// ---- DUTs/IO/Topology/Term_294_EK1100_DFE2A59E.TcDUT
{attribute 'GeneratedUsingTerminal: EK1100-0000-0018'}
{attribute addProperty BoxType "EK1100-0000-0018"}
{attribute addProperty Id "Term_300_EL1809EL1809_32157CFD20Term_304_EL2008EL2008_E2806B9511Term_305_EL2008EL2008_E2806B9511"}
{attribute addProperty CRC "3756172702"}
{attribute addProperty Size "42"}
{attribute addProperty Name "Term 294 (EK1100)"}
TYPE Term_294_EK1100_DFE2A59E EXTENDS EK1100_1FC0878B :
STRUCT
    {attribute addProperty Name "Term 300 (EL1809)"}
    {attribute addProperty PreviousPort "Term 294 (EK1100) : B"}
    {attribute addProperty SyncUnit "default"}
    Term_300_EL1809 : EL1809_32157CFD;
    {attribute addProperty Name "Term 304 (EL2008)"}
    {attribute addProperty PreviousPort "Term 300 (EL1809) : B"}
    {attribute addProperty SyncUnit "default"}
    Term_304_EL2008 : EL2008_E2806B95;
    {attribute addProperty Name "Term 305 (EL2008)"}
    {attribute addProperty PreviousPort "Term 304 (EL2008) : B"}
    {attribute addProperty SyncUnit "default"}
    Term_305_EL2008 : EL2008_E2806B95;
END_STRUCT
END_TYPE

// ---- DUTs/IO/Topology/Term_331_EK1100_B9C4E092.TcDUT
{attribute 'GeneratedUsingTerminal: EK1100-0000-0018'}
{attribute addProperty BoxType "EK1100-0000-0018"}
{attribute addProperty Id "Term_332_EL1809EL1809_32157CFD20"}
{attribute addProperty CRC "3116687506"}
{attribute addProperty Size "20"}
{attribute addProperty Name "Term 331 (EK1100)"}
TYPE Term_331_EK1100_B9C4E092 EXTENDS EK1100_1FC0878B :
STRUCT
    {attribute addProperty Name "Term 332 (EL1809)"}
    {attribute addProperty PreviousPort "Term 331 (EK1100) : B"}
    {attribute addProperty SyncUnit "default"}
    Term_332_EL1809 : EL1809_32157CFD;
END_STRUCT
END_TYPE

// ---- DUTs/IO/Topology/Term_333_EK1100_1D6F2042.TcDUT
{attribute 'GeneratedUsingTerminal: EK1100-0000-0018'}
{attribute addProperty BoxType "EK1100-0000-0018"}
{attribute addProperty Id "Term_334_EL1809EL1809_32157CFD20"}
{attribute addProperty CRC "493822018"}
{attribute addProperty Size "20"}
{attribute addProperty Name "Term 333 (EK1100)"}
TYPE Term_333_EK1100_1D6F2042 EXTENDS EK1100_1FC0878B :
STRUCT
    {attribute addProperty Name "Term 334 (EL1809)"}
    {attribute addProperty PreviousPort "Term 333 (EK1100) : B"}
    {attribute addProperty SyncUnit "default"}
    Term_334_EL1809 : EL1809_32157CFD;
END_STRUCT
END_TYPE

// ---- DUTs/IO/Topology/Term_330_EK1122_0EDE60FE.TcDUT
{attribute 'GeneratedUsingTerminal: EK1122-0000-0018'}
{attribute addProperty BoxType "EK1122-0000-0018"}
{attribute addProperty Id "Term_331_EK1100Term_331_EK1100_B9C4E09220Term_333_EK1100Term_333_EK1100_1D6F204220"}
{attribute addProperty CRC "249454846"}
{attribute addProperty Size "40"}
{attribute addProperty Name "Term 330 (EK1122)"}
TYPE Term_330_EK1122_0EDE60FE EXTENDS EK1122_1FC0878B :
STRUCT
    {attribute addProperty Name "Term 331 (EK1100)"}
    {attribute addProperty PreviousPort "Term 330 (EK1122) : D"}
    {attribute addProperty SyncUnit "default"}
    Term_331_EK1100 : Term_331_EK1100_B9C4E092;
    {attribute addProperty Name "Term 333 (EK1100)"}
    {attribute addProperty PreviousPort "Term 331 (EK1100) : C"}
    {attribute addProperty SyncUnit "default"}
    Term_333_EK1100 : Term_333_EK1100_1D6F2042;
END_STRUCT
END_TYPE

// ---- DUTs/IO/Topology/Term_307_EK1100_EB8FAA41.TcDUT
{attribute 'GeneratedUsingTerminal: EK1100-0000-0018'}
{attribute addProperty BoxType "EK1100-0000-0018"}
{attribute addProperty Id "Term_330_EK1122Term_330_EK1122_0EDE60FE40Term_335_EL2008EL2008_E2806B9511Term_336_EL2008EL2008_E2806B9511"}
{attribute addProperty CRC "3952060993"}
{attribute addProperty Size "62"}
{attribute addProperty Name "Term 307 (EK1100)"}
TYPE Term_307_EK1100_EB8FAA41 EXTENDS EK1100_1FC0878B :
STRUCT
    {attribute addProperty Name "Term 330 (EK1122)"}
    {attribute addProperty PreviousPort "Term 307 (EK1100) : B"}
    {attribute addProperty SyncUnit "default"}
    Term_330_EK1122 : Term_330_EK1122_0EDE60FE;
    {attribute addProperty Name "Term 335 (EL2008)"}
    {attribute addProperty PreviousPort "Term 330 (EK1122) : C"}
    {attribute addProperty SyncUnit "default"}
    Term_335_EL2008 : EL2008_E2806B95;
    {attribute addProperty Name "Term 336 (EL2008)"}
    {attribute addProperty PreviousPort "Term 335 (EL2008) : B"}
    {attribute addProperty SyncUnit "default"}
    Term_336_EL2008 : EL2008_E2806B95;
END_STRUCT
END_TYPE

// ---- DUTs/IO/Topology/Term_288_EK1122_18F8921F.TcDUT
{attribute 'GeneratedUsingTerminal: EK1122-0000-0018'}
{attribute addProperty BoxType "EK1122-0000-0018"}
{attribute addProperty Id "Term_289_EK1100Term_289_EK1100_9C677E5049Term_294_EK1100Term_294_EK1100_DFE2A59E42Term_307_EK1100Term_307_EK1100_EB8FAA4162"}
{attribute addProperty CRC "418943519"}
{attribute addProperty Size "153"}
{attribute addProperty Name "Term 288 (EK1122)"}
TYPE Term_288_EK1122_18F8921F EXTENDS EK1122_1FC0878B :
STRUCT
    {attribute addProperty Name "Term 289 (EK1100)"}
    {attribute addProperty PreviousPort "Term 288 (EK1122) : D"}
    {attribute addProperty SyncUnit "default"}
    Term_289_EK1100 : Term_289_EK1100_9C677E50;
    {attribute addProperty Name "Term 294 (EK1100)"}
    {attribute addProperty PreviousPort "Term 289 (EK1100) : C"}
    {attribute addProperty SyncUnit "default"}
    Term_294_EK1100 : Term_294_EK1100_DFE2A59E;
    {attribute addProperty Name "Term 307 (EK1100)"}
    {attribute addProperty PreviousPort "Term 294 (EK1100) : C"}
    {attribute addProperty SyncUnit "default"}
    Term_307_EK1100 : Term_307_EK1100_EB8FAA41;
END_STRUCT
END_TYPE

// ---- DUTs/IO/Topology/Term_146_EK1100_439F5464.TcDUT
{attribute 'GeneratedUsingTerminal: EK1100-0000-0018'}
{attribute addProperty BoxType "EK1100-0000-0018"}
{attribute addProperty Id "Term_147_EK1122Term_147_EK1122_CA6A5D16124Term_186_EK1122Term_186_EK1122_75C79D52124Term_148_EL1809EL1809_32157CFD20Term_149_EL1809EL1809_32157CFD20Term_150_EL1809EL1809_32157CFD20Term_151_EL1809EL1809_32157CFD20Term_152_EL1809EL1809_32157CFD20Term_288_EK1122Term_288_EK1122_18F8921F153Term_1158_EL2008EL2008_E2806B9511Term_1159_EL2008EL2008_E2806B9511Term_1160_EL2008EL2008_E2806B9511Term_1161_EL2008EL2008_E2806B9511Term_1162_EL2008EL2008_E2806B9511Term_1163_EL2008EL2008_E2806B9511"}
{attribute addProperty CRC "1134515300"}
{attribute addProperty Size "567"}
{attribute addProperty Name "Term 146 (EK1100)"}
TYPE Term_146_EK1100_439F5464 EXTENDS EK1100_1FC0878B :
STRUCT
    {attribute addProperty Name "Term 147 (EK1122)"}
    {attribute addProperty PreviousPort "Term 146 (EK1100) : B"}
    {attribute addProperty SyncUnit "default"}
    Term_147_EK1122 : Term_147_EK1122_CA6A5D16;
    {attribute addProperty Name "Term 186 (EK1122)"}
    {attribute addProperty PreviousPort "Term 147 (EK1122) : C"}
    {attribute addProperty SyncUnit "default"}
    Term_186_EK1122 : Term_186_EK1122_75C79D52;
    {attribute addProperty Name "Term 148 (EL1809)"}
    {attribute addProperty PreviousPort "Term 186 (EK1122) : C"}
    {attribute addProperty SyncUnit "default"}
    Term_148_EL1809 : EL1809_32157CFD;
    {attribute addProperty Name "Term 149 (EL1809)"}
    {attribute addProperty PreviousPort "Term 148 (EL1809) : B"}
    {attribute addProperty SyncUnit "default"}
    Term_149_EL1809 : EL1809_32157CFD;
    {attribute addProperty Name "Term 150 (EL1809)"}
    {attribute addProperty PreviousPort "Term 149 (EL1809) : B"}
    {attribute addProperty SyncUnit "default"}
    Term_150_EL1809 : EL1809_32157CFD;
    {attribute addProperty Name "Term 151 (EL1809)"}
    {attribute addProperty PreviousPort "Term 150 (EL1809) : B"}
    {attribute addProperty SyncUnit "default"}
    Term_151_EL1809 : EL1809_32157CFD;
    {attribute addProperty Name "Term 152 (EL1809)"}
    {attribute addProperty PreviousPort "Term 151 (EL1809) : B"}
    {attribute addProperty SyncUnit "default"}
    Term_152_EL1809 : EL1809_32157CFD;
    {attribute addProperty Name "Term 288 (EK1122)"}
    {attribute addProperty PreviousPort "Term 152 (EL1809) : B"}
    {attribute addProperty SyncUnit "default"}
    Term_288_EK1122 : Term_288_EK1122_18F8921F;
    {attribute addProperty Name "Term 1158 (EL2008)"}
    {attribute addProperty PreviousPort "Term 288 (EK1122) : C"}
    {attribute addProperty SyncUnit "default"}
    Term_1158_EL2008 : EL2008_E2806B95;
    {attribute addProperty Name "Term 1159 (EL2008)"}
    {attribute addProperty PreviousPort "Term 1158 (EL2008) : B"}
    {attribute addProperty SyncUnit "default"}
    Term_1159_EL2008 : EL2008_E2806B95;
    {attribute addProperty Name "Term 1160 (EL2008)"}
    {attribute addProperty PreviousPort "Term 1159 (EL2008) : B"}
    {attribute addProperty SyncUnit "default"}
    Term_1160_EL2008 : EL2008_E2806B95;
    {attribute addProperty Name "Term 1161 (EL2008)"}
    {attribute addProperty PreviousPort "Term 1160 (EL2008) : B"}
    {attribute addProperty SyncUnit "default"}
    Term_1161_EL2008 : EL2008_E2806B95;
    {attribute addProperty Name "Term 1162 (EL2008)"}
    {attribute addProperty PreviousPort "Term 1161 (EL2008) : B"}
    {attribute addProperty SyncUnit "default"}
    Term_1162_EL2008 : EL2008_E2806B95;
    {attribute addProperty Name "Term 1163 (EL2008)"}
    {attribute addProperty PreviousPort "Term 1162 (EL2008) : B"}
    {attribute addProperty SyncUnit "default"}
    Term_1163_EL2008 : EL2008_E2806B95;
END_STRUCT
END_TYPE

// ---- DUTs/IO/Topology/Device_3_EtherCAT_368E547E.TcDUT
{attribute 'GeneratedUsingTerminal: IODEVICETYPE_ETHERCATPROT'}
{attribute addProperty BoxType "IODEVICETYPE_ETHERCATPROT"}
{attribute addProperty Id "Term_146_EK1100Term_146_EK1100_439F5464567SyncUnitsSyncUnits_C3A34B5018InputsInputs_A65FACA410OutputsOutputs_23C0ED1D6InfoDataInfoData_84133AC922"}
{attribute addProperty CRC "915297406"}
{attribute addProperty Size "623"}
{attribute addProperty Name "Device 3 (EtherCAT)"}
TYPE Device_3_EtherCAT_368E547E EXTENDS TcoIo.EtcMasterBase_62654B43 :
STRUCT
    {attribute addProperty Name "Term 146 (EK1100)"}
    {attribute addProperty PreviousPort "Device 3 (EtherCAT) : Master"}
    {attribute addProperty SyncUnit "default"}
    Term_146_EK1100 : Term_146_EK1100_439F5464;
    {attribute addProperty Name "SyncUnits"}
    SyncUnits : SyncUnits_C3A34B50;
    {attribute addProperty Name "Inputs"}
    Inputs : TcoIo.Inputs_A65FACA4;
    {attribute addProperty Name "Outputs"}
    Outputs : TcoIo.Outputs_23C0ED1D;
    {attribute addProperty Name "InfoData"}
    InfoData : TcoIo.InfoData_84133AC9;
END_STRUCT
END_TYPE

// ---- DUTs/IO/Topology/R1_A2_EC_EK1122_F4361AFD.TcDUT
{attribute 'GeneratedUsingTerminal: EK1122-0000-0018'}
{attribute addProperty BoxType "EK1122-0000-0018"}
{attribute addProperty Id "Servo_A10_1_AX5106_0000_0203AX5106_1BD22F5129Servo_A10_2_AX5106_0000_0203AX5106_1BD22F5129Servo_A10_3_AX5106_0000_0203AX5106_1BD22F5129"}
{attribute addProperty CRC "4097186557"}
{attribute addProperty Size "87"}
{attribute addProperty Name "R1_A2_EC (EK1122)"}
TYPE R1_A2_EC_EK1122_F4361AFD EXTENDS EK1122_1FC0878B :
STRUCT
    {attribute addProperty Name "Servo_A10_1 (AX5106-0000-0203)"}
    {attribute addProperty PreviousPort "R1_A2_EC (EK1122) : D"}
    {attribute addProperty SyncUnit "default"}
    Servo_A10_1_AX5106_0000_0203 : AX5106_1BD22F51;
    {attribute addProperty Name "Servo_A10_2 (AX5106-0000-0203)"}
    {attribute addProperty PreviousPort "Servo_A10_1 (AX5106-0000-0203) : B"}
    {attribute addProperty SyncUnit "default"}
    Servo_A10_2_AX5106_0000_0203 : AX5106_1BD22F51;
    {attribute addProperty Name "Servo_A10_3 (AX5106-0000-0203)"}
    {attribute addProperty PreviousPort "Servo_A10_2 (AX5106-0000-0203) : B"}
    {attribute addProperty SyncUnit "default"}
    Servo_A10_3_AX5106_0000_0203 : AX5106_1BD22F51;
END_STRUCT
END_TYPE

// ---- DUTs/IO/Topology/R1_A3_EC_EK1122_981C12E1.TcDUT
{attribute 'GeneratedUsingTerminal: EK1122-0000-0018'}
{attribute addProperty BoxType "EK1122-0000-0018"}
{attribute addProperty Id "VI_2_AES_D_BC_ECAT_xAES_A3B0707168VI_4_AES_D_BC_ECAT_xAES_A3B0707168"}
{attribute addProperty CRC "2551976673"}
{attribute addProperty Size "136"}
{attribute addProperty Name "R1_A3_EC (EK1122)"}
TYPE R1_A3_EC_EK1122_981C12E1 EXTENDS EK1122_1FC0878B :
STRUCT
    {attribute addProperty Name "VI-2 (AES-D-BC-ECAT)"}
    {attribute addProperty PreviousPort "R1_A3_EC (EK1122) : D"}
    {attribute addProperty SyncUnit "default"}
    VI_2_AES_D_BC_ECAT_x : AES_A3B07071;
    {attribute addProperty Name "VI-4 (AES-D-BC-ECAT)"}
    {attribute addProperty PreviousPort "R1_A3_EC (EK1122) : B"}
    {attribute addProperty SyncUnit "default"}
    VI_4_AES_D_BC_ECAT_x : AES_A3B07071;
END_STRUCT
END_TYPE

// ---- DUTs/IO/Topology/R1_A4_X1_EK1100_C601B400.TcDUT
{attribute 'GeneratedUsingTerminal: EK1100-0000-0018'}
{attribute addProperty BoxType "EK1100-0000-0018"}
{attribute addProperty Id "R1_A4_X1_PN_EL6631EL6631_A0EC075C2R1_A4_X1_IA1_EL1809EL1809_32157CFD20R1_A4_X1_IA2_EL1809EL1809_32157CFD20R1_A4_X1_IA3_EL1809EL1809_32157CFD20R1_A4_X1_IA4_EL1809EL1809_32157CFD20R1_A4_X1_QA1_EL2809EL2809_2B6483BD19R1_A4_X1_QA2_EL2809EL2809_2B6483BD19R1_A4_X1_QA3_EL2809EL2809_2B6483BD19R1_A4_X1_EndTerminal_EL9010EL9010_D29C20850"}
{attribute addProperty CRC "3322000384"}
{attribute addProperty Size "139"}
{attribute addProperty Name "R1_A4_X1 (EK1100)"}
TYPE R1_A4_X1_EK1100_C601B400 EXTENDS EK1100_1FC0878B :
STRUCT
    {attribute addProperty Name "R1_A4_X1_PN (EL6631)"}
    {attribute addProperty PreviousPort "R1_A4_X1 (EK1100) : B"}
    {attribute addProperty SyncUnit "N10"}
    R1_A4_X1_PN_EL6631 : EL6631_A0EC075C;
    {attribute addProperty Name "R1_A4_X1_IA1 (EL1809)"}
    {attribute addProperty PreviousPort "R1_A4_X1_PN (EL6631) : B"}
    {attribute addProperty SyncUnit "N10"}
    R1_A4_X1_IA1_EL1809 : EL1809_32157CFD;
    {attribute addProperty Name "R1_A4_X1_IA2 (EL1809)"}
    {attribute addProperty PreviousPort "R1_A4_X1_IA1 (EL1809) : B"}
    {attribute addProperty SyncUnit "N10"}
    R1_A4_X1_IA2_EL1809 : EL1809_32157CFD;
    {attribute addProperty Name "R1_A4_X1_IA3 (EL1809)"}
    {attribute addProperty PreviousPort "R1_A4_X1_IA2 (EL1809) : B"}
    {attribute addProperty SyncUnit "N10"}
    R1_A4_X1_IA3_EL1809 : EL1809_32157CFD;
    {attribute addProperty Name "R1_A4_X1_IA4 (EL1809)"}
    {attribute addProperty PreviousPort "R1_A4_X1_IA3 (EL1809) : B"}
    {attribute addProperty SyncUnit "N10"}
    R1_A4_X1_IA4_EL1809 : EL1809_32157CFD;
    {attribute addProperty Name "R1_A4_X1_QA1 (EL2809)"}
    {attribute addProperty PreviousPort "R1_A4_X1_IA4 (EL1809) : B"}
    {attribute addProperty SyncUnit "N10"}
    R1_A4_X1_QA1_EL2809 : EL2809_2B6483BD;
    {attribute addProperty Name "R1_A4_X1_QA2 (EL2809)"}
    {attribute addProperty PreviousPort "R1_A4_X1_QA1 (EL2809) : B"}
    {attribute addProperty SyncUnit "N10"}
    R1_A4_X1_QA2_EL2809 : EL2809_2B6483BD;
    {attribute addProperty Name "R1_A4_X1_QA3 (EL2809)"}
    {attribute addProperty PreviousPort "R1_A4_X1_QA2 (EL2809) : B"}
    {attribute addProperty SyncUnit "N10"}
    R1_A4_X1_QA3_EL2809 : EL2809_2B6483BD;
    {attribute addProperty Name "R1_A4_X1_EndTerminal (EL9010)"}
    {attribute addProperty PreviousPort "R1_A4_X1_QA3 (EL2809) : B"}
    {attribute addProperty SyncUnit "default"}
    R1_A4_X1_EndTerminal_EL9010 : EL9010_D29C2085;
END_STRUCT
END_TYPE

// ---- DUTs/IO/Topology/R1_A4_X2_A2_EK1122_39ABCC27.TcDUT
{attribute 'GeneratedUsingTerminal: EK1122-0000-0018'}
{attribute addProperty BoxType "EK1122-0000-0018"}
{attribute addProperty Id "R1_A4_X2_A2_VI1_AES_D_BC_ECAT_xAES_B47A261080REX_350_IMecat_xIMecat_x_75C6CB6B170"}
{attribute addProperty CRC "967560231"}
{attribute addProperty Size "250"}
{attribute addProperty Name "R1_A4_X2_A2 (EK1122)"}
TYPE R1_A4_X2_A2_EK1122_39ABCC27 EXTENDS EK1122_1FC0878B :
STRUCT
    {attribute addProperty Name "R1_A4_X2_A2_VI1 (AES-D-BC-ECAT)"}
    {attribute addProperty PreviousPort "R1_A4_X2_A2 (EK1122) : D"}
    {attribute addProperty SyncUnit "S10"}
    R1_A4_X2_A2_VI1_AES_D_BC_ECAT_x : AES_B47A2610;
    {attribute addProperty Name "REX_350 (IMecat)"}
    {attribute addProperty PreviousPort "R1_A4_X2_A2 (EK1122) : B"}
    {attribute addProperty SyncUnit "default"}
    REX_350_IMecat_x : IMecat_x_75C6CB6B;
END_STRUCT
END_TYPE

// ---- DUTs/IO/Topology/R1_A4_X2_EK1100_6F5FB3BA.TcDUT
{attribute 'GeneratedUsingTerminal: EK1100-0000-0018'}
{attribute addProperty BoxType "EK1100-0000-0018"}
{attribute addProperty Id "R1_A4_X2_A2_EK1122R1_A4_X2_A2_EK1122_39ABCC27250R1_A4_X2_IA1_EL1809EL1809_32157CFD20R1_A4_X2_IA2_EL1809EL1809_32157CFD20R1_A4_X2_IA3_EL1809EL1809_32157CFD20R1_A4_X2_IA4_EL1809EL1809_32157CFD20R1_A4_X2_IA5_EL1809EL1809_32157CFD20R1_A4_X2_QA1_EL2809EL2809_2B6483BD19R1_A4_X2_QA2_EL2809EL2809_2B6483BD19R1_A4_X2_QA3_EL2809EL2809_2B6483BD19R1_A4_X2_EndTerminal_EL9010EL9010_D29C20850"}
{attribute addProperty CRC "1868542906"}
{attribute addProperty Size "407"}
{attribute addProperty Name "R1_A4_X2 (EK1100)"}
TYPE R1_A4_X2_EK1100_6F5FB3BA EXTENDS EK1100_1FC0878B :
STRUCT
    {attribute addProperty Name "R1_A4_X2_A2 (EK1122)"}
    {attribute addProperty PreviousPort "R1_A4_X2 (EK1100) : B"}
    {attribute addProperty SyncUnit "default"}
    R1_A4_X2_A2_EK1122 : R1_A4_X2_A2_EK1122_39ABCC27;
    {attribute addProperty Name "R1_A4_X2_IA1 (EL1809)"}
    {attribute addProperty PreviousPort "R1_A4_X2_A2 (EK1122) : C"}
    {attribute addProperty SyncUnit "S10"}
    R1_A4_X2_IA1_EL1809 : EL1809_32157CFD;
    {attribute addProperty Name "R1_A4_X2_IA2 (EL1809)"}
    {attribute addProperty PreviousPort "R1_A4_X2_IA1 (EL1809) : B"}
    {attribute addProperty SyncUnit "S10"}
    R1_A4_X2_IA2_EL1809 : EL1809_32157CFD;
    {attribute addProperty Name "R1_A4_X2_IA3 (EL1809)"}
    {attribute addProperty PreviousPort "R1_A4_X2_IA2 (EL1809) : B"}
    {attribute addProperty SyncUnit "S10"}
    R1_A4_X2_IA3_EL1809 : EL1809_32157CFD;
    {attribute addProperty Name "R1_A4_X2_IA4 (EL1809)"}
    {attribute addProperty PreviousPort "R1_A4_X2_IA3 (EL1809) : B"}
    {attribute addProperty SyncUnit "S10"}
    R1_A4_X2_IA4_EL1809 : EL1809_32157CFD;
    {attribute addProperty Name "R1_A4_X2_IA5 (EL1809)"}
    {attribute addProperty PreviousPort "R1_A4_X2_IA4 (EL1809) : B"}
    {attribute addProperty SyncUnit "S10"}
    R1_A4_X2_IA5_EL1809 : EL1809_32157CFD;
    {attribute addProperty Name "R1_A4_X2_QA1 (EL2809)"}
    {attribute addProperty PreviousPort "R1_A4_X2_IA5 (EL1809) : B"}
    {attribute addProperty SyncUnit "S10"}
    R1_A4_X2_QA1_EL2809 : EL2809_2B6483BD;
    {attribute addProperty Name "R1_A4_X2_QA2 (EL2809)"}
    {attribute addProperty PreviousPort "R1_A4_X2_QA1 (EL2809) : B"}
    {attribute addProperty SyncUnit "S10"}
    R1_A4_X2_QA2_EL2809 : EL2809_2B6483BD;
    {attribute addProperty Name "R1_A4_X2_QA3 (EL2809)"}
    {attribute addProperty PreviousPort "R1_A4_X2_QA2 (EL2809) : B"}
    {attribute addProperty SyncUnit "S10"}
    R1_A4_X2_QA3_EL2809 : EL2809_2B6483BD;
    {attribute addProperty Name "R1_A4_X2_EndTerminal (EL9010)"}
    {attribute addProperty PreviousPort "R1_A4_X2_QA3 (EL2809) : B"}
    {attribute addProperty SyncUnit "default"}
    R1_A4_X2_EndTerminal_EL9010 : EL9010_D29C2085;
END_STRUCT
END_TYPE

// ---- DUTs/IO/Topology/R1_A4_EC_EK1122_467C5A0B.TcDUT
{attribute 'GeneratedUsingTerminal: EK1122-0000-0018'}
{attribute addProperty BoxType "EK1122-0000-0018"}
{attribute addProperty Id "R1_A4_X1_EK1100R1_A4_X1_EK1100_C601B400139R1_A4_X2_EK1100R1_A4_X2_EK1100_6F5FB3BA407"}
{attribute addProperty CRC "1182554635"}
{attribute addProperty Size "546"}
{attribute addProperty Name "R1_A4_EC (EK1122)"}
TYPE R1_A4_EC_EK1122_467C5A0B EXTENDS EK1122_1FC0878B :
STRUCT
    {attribute addProperty Name "R1_A4_X1 (EK1100)"}
    {attribute addProperty PreviousPort "R1_A4_EC (EK1122) : D"}
    {attribute addProperty SyncUnit "default"}
    R1_A4_X1_EK1100 : R1_A4_X1_EK1100_C601B400;
    {attribute addProperty Name "R1_A4_X2 (EK1100)"}
    {attribute addProperty PreviousPort "R1_A4_EC (EK1122) : B"}
    {attribute addProperty SyncUnit "default"}
    R1_A4_X2_EK1100 : R1_A4_X2_EK1100_6F5FB3BA;
END_STRUCT
END_TYPE

// ---- DUTs/IO/Topology/R1_EK1100_4AD22B7B.TcDUT
{attribute 'GeneratedUsingTerminal: EK1100-0000-0018'}
{attribute addProperty BoxType "EK1100-0000-0018"}
{attribute addProperty Id "R1_A2_EC_EK1122R1_A2_EC_EK1122_F4361AFD87R1_A3_EC_EK1122R1_A3_EC_EK1122_981C12E1136R1_A4_EC_EK1122R1_A4_EC_EK1122_467C5A0B546R1_A5_DI_EL1809EL1809_32157CFD20R1_A6_DI_EL1809EL1809_32157CFD20R1_A7_DI_EL1809EL1809_32157CFD20R1_A8_DI_EL1809EL1809_32157CFD20R1_A9_DI_EL1809EL1809_32157CFD20R1_A10_DI_EL1809EL1809_32157CFD20R1_A11_DI_EL1809EL1809_32157CFD20R1_A12_DI_EL1809EL1809_32157CFD20R1_A13_DI_EL1809EL1809_32157CFD20R1_A14_DI_EL1809EL1809_32157CFD20R1_A15_DI_EL1809EL1809_32157CFD20R1_A16_DI_EL1809EL1809_32157CFD20R1_A17_DI_EL1809EL1809_32157CFD20R1_A18_DO_EL2809EL2809_2B6483BD19R1_A19_DO_EL2809EL2809_2B6483BD19R1_A20_DO_EL2809EL2809_2B6483BD19R1_A21_DO_EL2809EL2809_2B6483BD19R1_A22_DO_EL2809EL2809_2B6483BD19R1_A23_DO_EL2809EL2809_2B6483BD19R1_EndTerminal_EL9011EL9011_D65D3D320"}
{attribute addProperty CRC "1255287675"}
{attribute addProperty Size "1143"}
{attribute addProperty Name "R1 (EK1100)"}
TYPE R1_EK1100_4AD22B7B EXTENDS EK1100_1FC0878B :
STRUCT
    {attribute addProperty Name "R1_A2_EC (EK1122)"}
    {attribute addProperty PreviousPort "R1 (EK1100) : B"}
    {attribute addProperty SyncUnit "default"}
    R1_A2_EC_EK1122 : R1_A2_EC_EK1122_F4361AFD;
    {attribute addProperty Name "R1_A3_EC (EK1122)"}
    {attribute addProperty PreviousPort "R1_A2_EC (EK1122) : C"}
    {attribute addProperty SyncUnit "default"}
    R1_A3_EC_EK1122 : R1_A3_EC_EK1122_981C12E1;
    {attribute addProperty Name "R1_A4_EC (EK1122)"}
    {attribute addProperty PreviousPort "R1_A3_EC (EK1122) : C"}
    {attribute addProperty SyncUnit "default"}
    R1_A4_EC_EK1122 : R1_A4_EC_EK1122_467C5A0B;
    {attribute addProperty Name "R1_A5_DI (EL1809)"}
    {attribute addProperty PreviousPort "R1_A4_EC (EK1122) : C"}
    {attribute addProperty SyncUnit "default"}
    R1_A5_DI_EL1809 : EL1809_32157CFD;
    {attribute addProperty Name "R1_A6_DI (EL1809)"}
    {attribute addProperty PreviousPort "R1_A5_DI (EL1809) : B"}
    {attribute addProperty SyncUnit "default"}
    R1_A6_DI_EL1809 : EL1809_32157CFD;
    {attribute addProperty Name "R1_A7_DI (EL1809)"}
    {attribute addProperty PreviousPort "R1_A6_DI (EL1809) : B"}
    {attribute addProperty SyncUnit "default"}
    R1_A7_DI_EL1809 : EL1809_32157CFD;
    {attribute addProperty Name "R1_A8_DI (EL1809)"}
    {attribute addProperty PreviousPort "R1_A7_DI (EL1809) : B"}
    {attribute addProperty SyncUnit "default"}
    R1_A8_DI_EL1809 : EL1809_32157CFD;
    {attribute addProperty Name "R1_A9_DI (EL1809)"}
    {attribute addProperty PreviousPort "R1_A8_DI (EL1809) : B"}
    {attribute addProperty SyncUnit "default"}
    R1_A9_DI_EL1809 : EL1809_32157CFD;
    {attribute addProperty Name "R1_A10_DI (EL1809)"}
    {attribute addProperty PreviousPort "R1_A9_DI (EL1809) : B"}
    {attribute addProperty SyncUnit "default"}
    R1_A10_DI_EL1809 : EL1809_32157CFD;
    {attribute addProperty Name "R1_A11_DI (EL1809)"}
    {attribute addProperty PreviousPort "R1_A10_DI (EL1809) : B"}
    {attribute addProperty SyncUnit "default"}
    R1_A11_DI_EL1809 : EL1809_32157CFD;
    {attribute addProperty Name "R1_A12_DI (EL1809)"}
    {attribute addProperty PreviousPort "R1_A11_DI (EL1809) : B"}
    {attribute addProperty SyncUnit "default"}
    R1_A12_DI_EL1809 : EL1809_32157CFD;
    {attribute addProperty Name "R1_A13_DI (EL1809)"}
    {attribute addProperty PreviousPort "R1_A12_DI (EL1809) : B"}
    {attribute addProperty SyncUnit "default"}
    R1_A13_DI_EL1809 : EL1809_32157CFD;
    {attribute addProperty Name "R1_A14_DI (EL1809)"}
    {attribute addProperty PreviousPort "R1_A13_DI (EL1809) : B"}
    {attribute addProperty SyncUnit "default"}
    R1_A14_DI_EL1809 : EL1809_32157CFD;
    {attribute addProperty Name "R1_A15_DI (EL1809)"}
    {attribute addProperty PreviousPort "R1_A14_DI (EL1809) : B"}
    {attribute addProperty SyncUnit "default"}
    R1_A15_DI_EL1809 : EL1809_32157CFD;
    {attribute addProperty Name "R1_A16_DI (EL1809)"}
    {attribute addProperty PreviousPort "R1_A15_DI (EL1809) : B"}
    {attribute addProperty SyncUnit "default"}
    R1_A16_DI_EL1809 : EL1809_32157CFD;
    {attribute addProperty Name "R1_A17_DI (EL1809)"}
    {attribute addProperty PreviousPort "R1_A16_DI (EL1809) : B"}
    {attribute addProperty SyncUnit "default"}
    R1_A17_DI_EL1809 : EL1809_32157CFD;
    {attribute addProperty Name "R1_A18_DO (EL2809)"}
    {attribute addProperty PreviousPort "R1_A17_DI (EL1809) : B"}
    {attribute addProperty SyncUnit "default"}
    R1_A18_DO_EL2809 : EL2809_2B6483BD;
    {attribute addProperty Name "R1_A19_DO (EL2809)"}
    {attribute addProperty PreviousPort "R1_A18_DO (EL2809) : B"}
    {attribute addProperty SyncUnit "default"}
    R1_A19_DO_EL2809 : EL2809_2B6483BD;
    {attribute addProperty Name "R1_A20_DO (EL2809)"}
    {attribute addProperty PreviousPort "R1_A19_DO (EL2809) : B"}
    {attribute addProperty SyncUnit "default"}
    R1_A20_DO_EL2809 : EL2809_2B6483BD;
    {attribute addProperty Name "R1_A21_DO (EL2809)"}
    {attribute addProperty PreviousPort "R1_A20_DO (EL2809) : B"}
    {attribute addProperty SyncUnit "default"}
    R1_A21_DO_EL2809 : EL2809_2B6483BD;
    {attribute addProperty Name "R1_A22_DO (EL2809)"}
    {attribute addProperty PreviousPort "R1_A21_DO (EL2809) : B"}
    {attribute addProperty SyncUnit "default"}
    R1_A22_DO_EL2809 : EL2809_2B6483BD;
    {attribute addProperty Name "R1_A23_DO (EL2809)"}
    {attribute addProperty PreviousPort "R1_A22_DO (EL2809) : B"}
    {attribute addProperty SyncUnit "default"}
    R1_A23_DO_EL2809 : EL2809_2B6483BD;
    {attribute addProperty Name "R1_EndTerminal (EL9011)"}
    {attribute addProperty PreviousPort "R1_A23_DO (EL2809) : B"}
    {attribute addProperty SyncUnit "default"}
    R1_EndTerminal_EL9011 : EL9011_D65D3D32;
END_STRUCT
END_TYPE

// ---- DUTs/IO/Topology/R2_A2_EC_EK1122_6D3594D4.TcDUT
{attribute 'GeneratedUsingTerminal: EK1122-0000-0018'}
{attribute addProperty BoxType "EK1122-0000-0018"}
{attribute addProperty Id "Servo_A20_2_AX5103_0000_0203AX5103_1BD22F5129VI_3_AES_D_BC_ECAT_xAES_A3B0707168"}
{attribute addProperty CRC "1832228052"}
{attribute addProperty Size "97"}
{attribute addProperty Name "R2_A2_EC (EK1122)"}
TYPE R2_A2_EC_EK1122_6D3594D4 EXTENDS EK1122_1FC0878B :
STRUCT
    {attribute addProperty Name "Servo_A20-2 (AX5103-0000-0203)"}
    {attribute addProperty PreviousPort "R2_A2_EC (EK1122) : D"}
    {attribute addProperty SyncUnit "default"}
    Servo_A20_2_AX5103_0000_0203 : AX5103_1BD22F51;
    {attribute addProperty Name "VI-3 (AES-D-BC-ECAT)"}
    {attribute addProperty PreviousPort "R2_A2_EC (EK1122) : B"}
    {attribute addProperty SyncUnit "default"}
    VI_3_AES_D_BC_ECAT_x : AES_A3B07071;
END_STRUCT
END_TYPE

// ---- DUTs/IO/Topology/R2_EK1100_10D8A594.TcDUT
{attribute 'GeneratedUsingTerminal: EK1100-0000-0018'}
{attribute addProperty BoxType "EK1100-0000-0018"}
{attribute addProperty Id "R2_A2_EC_EK1122R2_A2_EC_EK1122_6D3594D497R2_A3_DI_EL1809EL1809_32157CFD20R2_A4_DI_EL1809EL1809_32157CFD20R2_A5_DI_EL1809EL1809_32157CFD20R2_A6_DI_EL1809EL1809_32157CFD20R2_A7_DI_EL1809EL1809_32157CFD20R2_A8_DI_EL1809EL1809_32157CFD20R2_A9_DI_EL1809EL1809_32157CFD20R2_A10_DI_EL1809EL1809_32157CFD20R2_A11_DC_EL7332EL7332_DFB2BED746R2_A12_DI_EL1809EL1809_32157CFD20R2_A13_DI_EL1809EL1809_32157CFD20R2_A14_DI_EL1809EL1809_32157CFD20R2_A15_DO_EL2809EL2809_2B6483BD19R2_A16_DO_EL2809EL2809_2B6483BD19R2_A17_DO_EL2809EL2809_2B6483BD19R2_A18_DO_EL2809EL2809_2B6483BD19R2_A19_DO_EL2809EL2809_2B6483BD19R2_EndTerminal_EL9011EL9011_D65D3D320"}
{attribute addProperty CRC "282633620"}
{attribute addProperty Size "458"}
{attribute addProperty Name "R2 (EK1100)"}
TYPE R2_EK1100_10D8A594 EXTENDS EK1100_1FC0878B :
STRUCT
    {attribute addProperty Name "R2_A2_EC (EK1122)"}
    {attribute addProperty PreviousPort "R2 (EK1100) : B"}
    {attribute addProperty SyncUnit "default"}
    R2_A2_EC_EK1122 : R2_A2_EC_EK1122_6D3594D4;
    {attribute addProperty Name "R2_A3_DI (EL1809)"}
    {attribute addProperty PreviousPort "R2_A2_EC (EK1122) : C"}
    {attribute addProperty SyncUnit "default"}
    R2_A3_DI_EL1809 : EL1809_32157CFD;
    {attribute addProperty Name "R2_A4_DI (EL1809)"}
    {attribute addProperty PreviousPort "R2_A3_DI (EL1809) : B"}
    {attribute addProperty SyncUnit "default"}
    R2_A4_DI_EL1809 : EL1809_32157CFD;
    {attribute addProperty Name "R2_A5_DI (EL1809)"}
    {attribute addProperty PreviousPort "R2_A4_DI (EL1809) : B"}
    {attribute addProperty SyncUnit "default"}
    R2_A5_DI_EL1809 : EL1809_32157CFD;
    {attribute addProperty Name "R2_A6_DI (EL1809)"}
    {attribute addProperty PreviousPort "R2_A5_DI (EL1809) : B"}
    {attribute addProperty SyncUnit "default"}
    R2_A6_DI_EL1809 : EL1809_32157CFD;
    {attribute addProperty Name "R2_A7_DI (EL1809)"}
    {attribute addProperty PreviousPort "R2_A6_DI (EL1809) : B"}
    {attribute addProperty SyncUnit "default"}
    R2_A7_DI_EL1809 : EL1809_32157CFD;
    {attribute addProperty Name "R2_A8_DI (EL1809)"}
    {attribute addProperty PreviousPort "R2_A7_DI (EL1809) : B"}
    {attribute addProperty SyncUnit "default"}
    R2_A8_DI_EL1809 : EL1809_32157CFD;
    {attribute addProperty Name "R2_A9_DI (EL1809)"}
    {attribute addProperty PreviousPort "R2_A8_DI (EL1809) : B"}
    {attribute addProperty SyncUnit "default"}
    R2_A9_DI_EL1809 : EL1809_32157CFD;
    {attribute addProperty Name "R2_A10_DI (EL1809)"}
    {attribute addProperty PreviousPort "R2_A9_DI (EL1809) : B"}
    {attribute addProperty SyncUnit "default"}
    R2_A10_DI_EL1809 : EL1809_32157CFD;
    {attribute addProperty Name "R2_A11_DC (EL7332)"}
    {attribute addProperty PreviousPort "R2_A10_DI (EL1809) : B"}
    {attribute addProperty SyncUnit "default"}
    R2_A11_DC_EL7332 : EL7332_DFB2BED7;
    {attribute addProperty Name "R2_A12_DI (EL1809)"}
    {attribute addProperty PreviousPort "R2_A11_DC (EL7332) : B"}
    {attribute addProperty SyncUnit "default"}
    R2_A12_DI_EL1809 : EL1809_32157CFD;
    {attribute addProperty Name "R2_A13_DI (EL1809)"}
    {attribute addProperty PreviousPort "R2_A12_DI (EL1809) : B"}
    {attribute addProperty SyncUnit "default"}
    R2_A13_DI_EL1809 : EL1809_32157CFD;
    {attribute addProperty Name "R2_A14_DI (EL1809)"}
    {attribute addProperty PreviousPort "R2_A13_DI (EL1809) : B"}
    {attribute addProperty SyncUnit "default"}
    R2_A14_DI_EL1809 : EL1809_32157CFD;
    {attribute addProperty Name "R2_A15_DO (EL2809)"}
    {attribute addProperty PreviousPort "R2_A14_DI (EL1809) : B"}
    {attribute addProperty SyncUnit "default"}
    R2_A15_DO_EL2809 : EL2809_2B6483BD;
    {attribute addProperty Name "R2_A16_DO (EL2809)"}
    {attribute addProperty PreviousPort "R2_A15_DO (EL2809) : B"}
    {attribute addProperty SyncUnit "default"}
    R2_A16_DO_EL2809 : EL2809_2B6483BD;
    {attribute addProperty Name "R2_A17_DO (EL2809)"}
    {attribute addProperty PreviousPort "R2_A16_DO (EL2809) : B"}
    {attribute addProperty SyncUnit "default"}
    R2_A17_DO_EL2809 : EL2809_2B6483BD;
    {attribute addProperty Name "R2_A18_DO (EL2809)"}
    {attribute addProperty PreviousPort "R2_A17_DO (EL2809) : B"}
    {attribute addProperty SyncUnit "default"}
    R2_A18_DO_EL2809 : EL2809_2B6483BD;
    {attribute addProperty Name "R2_A19_DO (EL2809)"}
    {attribute addProperty PreviousPort "R2_A18_DO (EL2809) : B"}
    {attribute addProperty SyncUnit "default"}
    R2_A19_DO_EL2809 : EL2809_2B6483BD;
    {attribute addProperty Name "R2_EndTerminal (EL9011)"}
    {attribute addProperty PreviousPort "R2_A19_DO (EL2809) : B"}
    {attribute addProperty SyncUnit "default"}
    R2_EndTerminal_EL9011 : EL9011_D65D3D32;
END_STRUCT
END_TYPE

// ---- DUTs/IO/Topology/R3_A2_EC_EK1122_9D59CDC8.TcDUT
{attribute 'GeneratedUsingTerminal: EK1122-0000-0018'}
{attribute addProperty BoxType "EK1122-0000-0018"}
{attribute addProperty Id "R3_FESTO_CMMP_AS_V4p0_CiA402CMMP_93B92D5237VI_1_AES_D_BC_ECAT_xAES_A3B0707168"}
{attribute addProperty CRC "2639908296"}
{attribute addProperty Size "105"}
{attribute addProperty Name "R3_A2_EC (EK1122)"}
TYPE R3_A2_EC_EK1122_9D59CDC8 EXTENDS EK1122_1FC0878B :
STRUCT
    {attribute addProperty Name "R3_FESTO (CMMP-AS V4p0 CiA402)"}
    {attribute addProperty PreviousPort "R3_A2_EC (EK1122) : D"}
    {attribute addProperty SyncUnit "default"}
    R3_FESTO_CMMP_AS_V4p0_CiA402 : CMMP_93B92D52;
    {attribute addProperty Name "VI-1 (AES-D-BC-ECAT)"}
    {attribute addProperty PreviousPort "R3_A2_EC (EK1122) : B"}
    {attribute addProperty SyncUnit "default"}
    VI_1_AES_D_BC_ECAT_x : AES_A3B07071;
END_STRUCT
END_TYPE

// ---- DUTs/IO/Topology/R3_EK1100_C7887D6C.TcDUT
{attribute 'GeneratedUsingTerminal: EK1100-0000-0018'}
{attribute addProperty BoxType "EK1100-0000-0018"}
{attribute addProperty Id "R3_A2_EC_EK1122R3_A2_EC_EK1122_9D59CDC8105R3_A3_DI_EL1809EL1809_32157CFD20R3_A4_DI_EL1809EL1809_32157CFD20R3_A5_DI_EL1809EL1809_32157CFD20R3_A6_DI_EL1809EL1809_32157CFD20R3_A7_DI_EL1809EL1809_32157CFD20R3_A8_DI_EL1809EL1809_32157CFD20R3_A9_DO_EL2809EL2809_2B6483BD19R3_A10_DO_EL2809EL2809_2B6483BD19R3_EndTerminal_EL9011EL9011_D65D3D320"}
{attribute addProperty CRC "3347610988"}
{attribute addProperty Size "263"}
{attribute addProperty Name "R3 (EK1100)"}
TYPE R3_EK1100_C7887D6C EXTENDS EK1100_1FC0878B :
STRUCT
    {attribute addProperty Name "R3_A2_EC (EK1122)"}
    {attribute addProperty PreviousPort "R3 (EK1100) : B"}
    {attribute addProperty SyncUnit "default"}
    R3_A2_EC_EK1122 : R3_A2_EC_EK1122_9D59CDC8;
    {attribute addProperty Name "R3_A3_DI (EL1809)"}
    {attribute addProperty PreviousPort "R3_A2_EC (EK1122) : C"}
    {attribute addProperty SyncUnit "default"}
    R3_A3_DI_EL1809 : EL1809_32157CFD;
    {attribute addProperty Name "R3_A4_DI (EL1809)"}
    {attribute addProperty PreviousPort "R3_A3_DI (EL1809) : B"}
    {attribute addProperty SyncUnit "default"}
    R3_A4_DI_EL1809 : EL1809_32157CFD;
    {attribute addProperty Name "R3_A5_DI (EL1809)"}
    {attribute addProperty PreviousPort "R3_A4_DI (EL1809) : B"}
    {attribute addProperty SyncUnit "default"}
    R3_A5_DI_EL1809 : EL1809_32157CFD;
    {attribute addProperty Name "R3_A6_DI (EL1809)"}
    {attribute addProperty PreviousPort "R3_A5_DI (EL1809) : B"}
    {attribute addProperty SyncUnit "default"}
    R3_A6_DI_EL1809 : EL1809_32157CFD;
    {attribute addProperty Name "R3_A7_DI (EL1809)"}
    {attribute addProperty PreviousPort "R3_A6_DI (EL1809) : B"}
    {attribute addProperty SyncUnit "default"}
    R3_A7_DI_EL1809 : EL1809_32157CFD;
    {attribute addProperty Name "R3_A8_DI (EL1809)"}
    {attribute addProperty PreviousPort "R3_A7_DI (EL1809) : B"}
    {attribute addProperty SyncUnit "default"}
    R3_A8_DI_EL1809 : EL1809_32157CFD;
    {attribute addProperty Name "R3_A9_DO (EL2809)"}
    {attribute addProperty PreviousPort "R3_A8_DI (EL1809) : B"}
    {attribute addProperty SyncUnit "default"}
    R3_A9_DO_EL2809 : EL2809_2B6483BD;
    {attribute addProperty Name "R3_A10_DO (EL2809)"}
    {attribute addProperty PreviousPort "R3_A9_DO (EL2809) : B"}
    {attribute addProperty SyncUnit "default"}
    R3_A10_DO_EL2809 : EL2809_2B6483BD;
    {attribute addProperty Name "R3_EndTerminal (EL9011)"}
    {attribute addProperty PreviousPort "R3_A10_DO (EL2809) : B"}
    {attribute addProperty SyncUnit "default"}
    R3_EndTerminal_EL9011 : EL9011_D65D3D32;
END_STRUCT
END_TYPE

// ---- DUTs/IO/Topology/RH_A2_X2_EK1100_67419BB1.TcDUT
{attribute 'GeneratedUsingTerminal: EK1100-0000-0018'}
{attribute addProperty BoxType "EK1100-0000-0018"}
{attribute addProperty Id "RH_A2_X2_A2_EL7211_0010EL7211_008D5C9A30RH_A2_X2_A3_EL1809EL1809_32157CFD20RH_A2_X2_A4_EL2809EL2809_2B6483BD19Term_1057_EL9011EL9011_D65D3D320"}
{attribute addProperty CRC "1732352945"}
{attribute addProperty Size "69"}
{attribute addProperty Name "RH_A2_X2 (EK1100)"}
TYPE RH_A2_X2_EK1100_67419BB1 EXTENDS EK1100_1FC0878B :
STRUCT
    {attribute addProperty Name "RH_A2_X2_A2 (EL7211-0010)"}
    {attribute addProperty PreviousPort "RH_A2_X2 (EK1100) : B"}
    {attribute addProperty SyncUnit "RH"}
    RH_A2_X2_A2_EL7211_0010 : EL7211_008D5C9A;
    {attribute addProperty Name "RH_A2_X2_A3 (EL1809)"}
    {attribute addProperty PreviousPort "RH_A2_X2_A2 (EL7211-0010) : B"}
    {attribute addProperty SyncUnit "RH"}
    RH_A2_X2_A3_EL1809 : EL1809_32157CFD;
    {attribute addProperty Name "RH_A2_X2_A4 (EL2809)"}
    {attribute addProperty PreviousPort "RH_A2_X2_A3 (EL1809) : B"}
    {attribute addProperty SyncUnit "RH"}
    RH_A2_X2_A4_EL2809 : EL2809_2B6483BD;
    {attribute addProperty Name "Term 1057 (EL9011)"}
    {attribute addProperty PreviousPort "RH_A2_X2_A4 (EL2809) : B"}
    {attribute addProperty SyncUnit "default"}
    Term_1057_EL9011 : EL9011_D65D3D32;
END_STRUCT
END_TYPE

// ---- DUTs/IO/Topology/RH_A2_EK1122_10728E09.TcDUT
{attribute 'GeneratedUsingTerminal: EK1122-0000-0018'}
{attribute addProperty BoxType "EK1122-0000-0018"}
{attribute addProperty Id "RH_SAFETY_Flexi_Gateway_GETC1Flexi_Gateway_GETC1_429ECB705RH_A2_X2_EK1100RH_A2_X2_EK1100_67419BB169"}
{attribute addProperty CRC "275942921"}
{attribute addProperty Size "74"}
{attribute addProperty Name "RH_A2 (EK1122)"}
TYPE RH_A2_EK1122_10728E09 EXTENDS EK1122_1FC0878B :
STRUCT
    {attribute addProperty Name "RH_SAFETY (Flexi Gateway GETC1)"}
    {attribute addProperty PreviousPort "RH_A2 (EK1122) : D"}
    {attribute addProperty SyncUnit "RH"}
    RH_SAFETY_Flexi_Gateway_GETC1 : Flexi_Gateway_GETC1_429ECB70;
    {attribute addProperty Name "RH_A2_X2 (EK1100)"}
    {attribute addProperty PreviousPort "RH_A2 (EK1122) : B"}
    {attribute addProperty SyncUnit "default"}
    RH_A2_X2_EK1100 : RH_A2_X2_EK1100_67419BB1;
END_STRUCT
END_TYPE

// ---- DUTs/IO/Topology/RH_EK1100_A5940DFE.TcDUT
{attribute 'GeneratedUsingTerminal: EK1100-0000-0018'}
{attribute addProperty BoxType "EK1100-0000-0018"}
{attribute addProperty Id "RH_A2_EK1122RH_A2_EK1122_10728E0974RH_A3_EL6631EL6631_A0EC075C2RH_A4_EL1809EL1809_32157CFD20RH_A5_EL1809EL1809_32157CFD20RH_A6_EL1809EL1809_32157CFD20RH_A7_EL2809EL2809_2B6483BD19RH_A8_EL1809EL1809_32157CFD20RH_A9_EL2809EL2809_2B6483BD19RH_A10_EL2809EL2809_2B6483BD19RH_A11_EL2809EL2809_2B6483BD19RH_EndTerminal_EL9011EL9011_D65D3D320"}
{attribute addProperty CRC "2777943550"}
{attribute addProperty Size "232"}
{attribute addProperty Name "RH (EK1100)"}
TYPE RH_EK1100_A5940DFE EXTENDS EK1100_1FC0878B :
STRUCT
    {attribute addProperty Name "RH_A2 (EK1122)"}
    {attribute addProperty PreviousPort "RH (EK1100) : B"}
    {attribute addProperty SyncUnit "default"}
    RH_A2_EK1122 : RH_A2_EK1122_10728E09;
    {attribute addProperty Name "RH_A3 (EL6631)"}
    {attribute addProperty PreviousPort "RH_A2 (EK1122) : C"}
    {attribute addProperty SyncUnit "RH"}
    RH_A3_EL6631 : EL6631_A0EC075C;
    {attribute addProperty Name "RH_A4 (EL1809)"}
    {attribute addProperty PreviousPort "RH_A3 (EL6631) : B"}
    {attribute addProperty SyncUnit "RH"}
    RH_A4_EL1809 : EL1809_32157CFD;
    {attribute addProperty Name "RH_A5 (EL1809)"}
    {attribute addProperty PreviousPort "RH_A4 (EL1809) : B"}
    {attribute addProperty SyncUnit "RH"}
    RH_A5_EL1809 : EL1809_32157CFD;
    {attribute addProperty Name "RH_A6 (EL1809)"}
    {attribute addProperty PreviousPort "RH_A5 (EL1809) : B"}
    {attribute addProperty SyncUnit "RH"}
    RH_A6_EL1809 : EL1809_32157CFD;
    {attribute addProperty Name "RH_A7 (EL2809)"}
    {attribute addProperty PreviousPort "RH_A6 (EL1809) : B"}
    {attribute addProperty SyncUnit "RH"}
    RH_A7_EL2809 : EL2809_2B6483BD;
    {attribute addProperty Name "RH_A8 (EL1809)"}
    {attribute addProperty PreviousPort "RH_A7 (EL2809) : B"}
    {attribute addProperty SyncUnit "RH"}
    RH_A8_EL1809 : EL1809_32157CFD;
    {attribute addProperty Name "RH_A9 (EL2809)"}
    {attribute addProperty PreviousPort "RH_A8 (EL1809) : B"}
    {attribute addProperty SyncUnit "RH"}
    RH_A9_EL2809 : EL2809_2B6483BD;
    {attribute addProperty Name "RH_A10 (EL2809)"}
    {attribute addProperty PreviousPort "RH_A9 (EL2809) : B"}
    {attribute addProperty SyncUnit "RH"}
    RH_A10_EL2809 : EL2809_2B6483BD;
    {attribute addProperty Name "RH_A11 (EL2809)"}
    {attribute addProperty PreviousPort "RH_A10 (EL2809) : B"}
    {attribute addProperty SyncUnit "RH"}
    RH_A11_EL2809 : EL2809_2B6483BD;
    {attribute addProperty Name "RH_EndTerminal (EL9011)"}
    {attribute addProperty PreviousPort "RH_A11 (EL2809) : B"}
    {attribute addProperty SyncUnit "default"}
    RH_EndTerminal_EL9011 : EL9011_D65D3D32;
END_STRUCT
END_TYPE

// ---- DUTs/IO/Topology/R4_A2_EC_EK1122_254454A1.TcDUT
{attribute 'GeneratedUsingTerminal: EK1122-0000-0018'}
{attribute addProperty BoxType "EK1122-0000-0018"}
{attribute addProperty Id "R4_FESTO_CMMP_AS_V4p0_CiA402CMMP_93B92D5237RH_EK1100RH_EK1100_A5940DFE232"}
{attribute addProperty CRC "625235105"}
{attribute addProperty Size "269"}
{attribute addProperty Name "R4_A2_EC (EK1122)"}
TYPE R4_A2_EC_EK1122_254454A1 EXTENDS EK1122_1FC0878B :
STRUCT
    {attribute addProperty Name "R4_FESTO (CMMP-AS V4p0 CiA402)"}
    {attribute addProperty PreviousPort "R4_A2_EC (EK1122) : D"}
    {attribute addProperty SyncUnit "default"}
    R4_FESTO_CMMP_AS_V4p0_CiA402 : CMMP_93B92D52;
    {attribute addProperty Name "RH (EK1100)"}
    {attribute addProperty PreviousPort "R4_A2_EC (EK1122) : B"}
    {attribute addProperty SyncUnit "default"}
    RH_EK1100 : RH_EK1100_A5940DFE;
END_STRUCT
END_TYPE

// ---- DUTs/IO/Topology/R4_EK1100_46A1248C.TcDUT
{attribute 'GeneratedUsingTerminal: EK1100-0000-0018'}
{attribute addProperty BoxType "EK1100-0000-0018"}
{attribute addProperty Id "R4_A2_EC_EK1122R4_A2_EC_EK1122_254454A1269R4_A3_DI_EL1809EL1809_32157CFD20R4_A4_DI_EL1809EL1809_32157CFD20R4_A5_DI_EL1809EL1809_32157CFD20R4_A6_DI_EL1809EL1809_32157CFD20R4_A7_DI_EL1809EL1809_32157CFD20R4_EndTerminal_EL9011EL9011_D65D3D320"}
{attribute addProperty CRC "1184965772"}
{attribute addProperty Size "369"}
{attribute addProperty Name "R4 (EK1100)"}
TYPE R4_EK1100_46A1248C EXTENDS EK1100_1FC0878B :
STRUCT
    {attribute addProperty Name "R4_A2_EC (EK1122)"}
    {attribute addProperty PreviousPort "R4 (EK1100) : B"}
    {attribute addProperty SyncUnit "default"}
    R4_A2_EC_EK1122 : R4_A2_EC_EK1122_254454A1;
    {attribute addProperty Name "R4_A3_DI (EL1809)"}
    {attribute addProperty PreviousPort "R4_A2_EC (EK1122) : C"}
    {attribute addProperty SyncUnit "default"}
    R4_A3_DI_EL1809 : EL1809_32157CFD;
    {attribute addProperty Name "R4_A4_DI (EL1809)"}
    {attribute addProperty PreviousPort "R4_A3_DI (EL1809) : B"}
    {attribute addProperty SyncUnit "default"}
    R4_A4_DI_EL1809 : EL1809_32157CFD;
    {attribute addProperty Name "R4_A5_DI (EL1809)"}
    {attribute addProperty PreviousPort "R4_A4_DI (EL1809) : B"}
    {attribute addProperty SyncUnit "default"}
    R4_A5_DI_EL1809 : EL1809_32157CFD;
    {attribute addProperty Name "R4_A6_DI (EL1809)"}
    {attribute addProperty PreviousPort "R4_A5_DI (EL1809) : B"}
    {attribute addProperty SyncUnit "default"}
    R4_A6_DI_EL1809 : EL1809_32157CFD;
    {attribute addProperty Name "R4_A7_DI (EL1809)"}
    {attribute addProperty PreviousPort "R4_A6_DI (EL1809) : B"}
    {attribute addProperty SyncUnit "default"}
    R4_A7_DI_EL1809 : EL1809_32157CFD;
    {attribute addProperty Name "R4_EndTerminal (EL9011)"}
    {attribute addProperty PreviousPort "R4_A7_DI (EL1809) : B"}
    {attribute addProperty SyncUnit "default"}
    R4_EndTerminal_EL9011 : EL9011_D65D3D32;
END_STRUCT
END_TYPE

// ---- DUTs/IO/Topology/A2_EK1122_967E4A9C.TcDUT
{attribute 'GeneratedUsingTerminal: EK1122-0000-0018'}
{attribute addProperty BoxType "EK1122-0000-0018"}
{attribute addProperty Id "VI_7_AES_D_BC_ECAT_xAES_A3B0707168"}
{attribute addProperty CRC "2524859036"}
{attribute addProperty Size "68"}
{attribute addProperty Name "A2 (EK1122)"}
TYPE A2_EK1122_967E4A9C EXTENDS EK1122_1FC0878B :
STRUCT
    {attribute addProperty Name "VI-7 (AES-D-BC-ECAT)"}
    {attribute addProperty PreviousPort "A2 (EK1122) : D"}
    {attribute addProperty SyncUnit "default"}
    VI_7_AES_D_BC_ECAT_x : AES_A3B07071;
END_STRUCT
END_TYPE

// ---- DUTs/IO/Topology/R4A_EK1100_48316913.TcDUT
{attribute 'GeneratedUsingTerminal: EK1100-0000-0018'}
{attribute addProperty BoxType "EK1100-0000-0018"}
{attribute addProperty Id "A2_EK1122A2_EK1122_967E4A9C68A3_EL1809EL1809_32157CFD20A4_EL1809EL1809_32157CFD20A5_EL1809EL1809_32157CFD20A6_EL1809EL1809_32157CFD20A7_EL3692EL3692_73B9410052A8_EL3692EL3692_73B9410052A9_EL2008EL2008_E2806B9511A10_EL2008EL2008_E2806B9511R4A_EndTerminal_EL9011EL9011_D65D3D320"}
{attribute addProperty CRC "1211197715"}
{attribute addProperty Size "274"}
{attribute addProperty Name "R4A (EK1100)"}
TYPE R4A_EK1100_48316913 EXTENDS EK1100_1FC0878B :
STRUCT
    {attribute addProperty Name "A2 (EK1122)"}
    {attribute addProperty PreviousPort "R4A (EK1100) : B"}
    {attribute addProperty SyncUnit "default"}
    A2_EK1122 : A2_EK1122_967E4A9C;
    {attribute addProperty Name "A3 (EL1809)"}
    {attribute addProperty PreviousPort "A2 (EK1122) : C"}
    {attribute addProperty SyncUnit "default"}
    A3_EL1809 : EL1809_32157CFD;
    {attribute addProperty Name "A4 (EL1809)"}
    {attribute addProperty PreviousPort "A3 (EL1809) : B"}
    {attribute addProperty SyncUnit "default"}
    A4_EL1809 : EL1809_32157CFD;
    {attribute addProperty Name "A5 (EL1809)"}
    {attribute addProperty PreviousPort "A4 (EL1809) : B"}
    {attribute addProperty SyncUnit "default"}
    A5_EL1809 : EL1809_32157CFD;
    {attribute addProperty Name "A6 (EL1809)"}
    {attribute addProperty PreviousPort "A5 (EL1809) : B"}
    {attribute addProperty SyncUnit "default"}
    A6_EL1809 : EL1809_32157CFD;
    {attribute addProperty Name "A7 (EL3692)"}
    {attribute addProperty PreviousPort "A6 (EL1809) : B"}
    {attribute addProperty SyncUnit "default"}
    A7_EL3692 : EL3692_73B94100;
    {attribute addProperty Name "A8 (EL3692)"}
    {attribute addProperty PreviousPort "A7 (EL3692) : B"}
    {attribute addProperty SyncUnit "default"}
    A8_EL3692 : EL3692_73B94100;
    {attribute addProperty Name "A9 (EL2008)"}
    {attribute addProperty PreviousPort "A8 (EL3692) : B"}
    {attribute addProperty SyncUnit "default"}
    A9_EL2008 : EL2008_E2806B95;
    {attribute addProperty Name "A10 (EL2008)"}
    {attribute addProperty PreviousPort "A9 (EL2008) : B"}
    {attribute addProperty SyncUnit "default"}
    A10_EL2008 : EL2008_E2806B95;
    {attribute addProperty Name "R4A_EndTerminal (EL9011)"}
    {attribute addProperty PreviousPort "A10 (EL2008) : B"}
    {attribute addProperty SyncUnit "default"}
    R4A_EndTerminal_EL9011 : EL9011_D65D3D32;
END_STRUCT
END_TYPE

// ---- DUTs/IO/Topology/R5_A2_EC_EK1122_D562526C.TcDUT
{attribute 'GeneratedUsingTerminal: EK1122-0000-0018'}
{attribute addProperty BoxType "EK1122-0000-0018"}
{attribute addProperty Id "VI_5_AES_D_BC_ECAT_xAES_A3B0707168"}
{attribute addProperty CRC "3579990636"}
{attribute addProperty Size "68"}
{attribute addProperty Name "R5_A2_EC (EK1122)"}
TYPE R5_A2_EC_EK1122_D562526C EXTENDS EK1122_1FC0878B :
STRUCT
    {attribute addProperty Name "VI-5 (AES-D-BC-ECAT)"}
    {attribute addProperty PreviousPort "R5_A2_EC (EK1122) : D"}
    {attribute addProperty SyncUnit "default"}
    VI_5_AES_D_BC_ECAT_x : AES_A3B07071;
END_STRUCT
END_TYPE

// ---- DUTs/IO/Topology/R5_EK1100_0007A337.TcDUT
{attribute 'GeneratedUsingTerminal: EK1100-0000-0018'}
{attribute addProperty BoxType "EK1100-0000-0018"}
{attribute addProperty Id "R5_A2_EC_EK1122R5_A2_EC_EK1122_D562526C68R5_A3_DI_EL1809EL1809_32157CFD20R5_A4_DI_EL1809EL1809_32157CFD20R5_A5_DO_EL2809EL2809_2B6483BD19R5_A6_DO_EL2809EL2809_2B6483BD19R5_EndTerminal_EL9011EL9011_D65D3D320"}
{attribute addProperty CRC "500535"}
{attribute addProperty Size "146"}
{attribute addProperty Name "R5 (EK1100)"}
TYPE R5_EK1100_0007A337 EXTENDS EK1100_1FC0878B :
STRUCT
    {attribute addProperty Name "R5_A2_EC (EK1122)"}
    {attribute addProperty PreviousPort "R5 (EK1100) : B"}
    {attribute addProperty SyncUnit "default"}
    R5_A2_EC_EK1122 : R5_A2_EC_EK1122_D562526C;
    {attribute addProperty Name "R5_A3_DI (EL1809)"}
    {attribute addProperty PreviousPort "R5_A2_EC (EK1122) : C"}
    {attribute addProperty SyncUnit "default"}
    R5_A3_DI_EL1809 : EL1809_32157CFD;
    {attribute addProperty Name "R5_A4_DI (EL1809)"}
    {attribute addProperty PreviousPort "R5_A3_DI (EL1809) : B"}
    {attribute addProperty SyncUnit "default"}
    R5_A4_DI_EL1809 : EL1809_32157CFD;
    {attribute addProperty Name "R5_A5_DO (EL2809)"}
    {attribute addProperty PreviousPort "R5_A4_DI (EL1809) : B"}
    {attribute addProperty SyncUnit "default"}
    R5_A5_DO_EL2809 : EL2809_2B6483BD;
    {attribute addProperty Name "R5_A6_DO (EL2809)"}
    {attribute addProperty PreviousPort "R5_A5_DO (EL2809) : B"}
    {attribute addProperty SyncUnit "default"}
    R5_A6_DO_EL2809 : EL2809_2B6483BD;
    {attribute addProperty Name "R5_EndTerminal (EL9011)"}
    {attribute addProperty PreviousPort "R5_A6_DO (EL2809) : B"}
    {attribute addProperty SyncUnit "default"}
    R5_EndTerminal_EL9011 : EL9011_D65D3D32;
END_STRUCT
END_TYPE

// ---- DUTs/IO/Topology/R6_EK1100_8C41F5F2.TcDUT
{attribute 'GeneratedUsingTerminal: EK1100-0000-0018'}
{attribute addProperty BoxType "EK1100-0000-0018"}
{attribute addProperty Id "R6_A2_DI_EL1809EL1809_32157CFD20R6_A3_DI_EL1809EL1809_32157CFD20R6_A4_DI_EL1809EL1809_32157CFD20R6_A5_DI_EL1809EL1809_32157CFD20R6_A6_DI_EL1809EL1809_32157CFD20R6_A7_DI_EL1809EL1809_32157CFD20R6_A8_DI_EL1809EL1809_32157CFD20R6_A9_DI_EL1809EL1809_32157CFD20R6_A10_DI_EL1809EL1809_32157CFD20R6_A11_DI_EL1809EL1809_32157CFD20R6_A12_DI_EL1809EL1809_32157CFD20R6_A13_DI_EL1809EL1809_32157CFD20R6_A14_DI_EL1809EL1809_32157CFD20R6_A15_DO_EL2809EL2809_2B6483BD19R6_A16_DO_EL2809EL2809_2B6483BD19R6_A17_DO_EL2809EL2809_2B6483BD19R6_A18_DO_EL2809EL2809_2B6483BD19R6_EndTerminal_EL9011EL9011_D65D3D320"}
{attribute addProperty CRC "2353133042"}
{attribute addProperty Size "336"}
{attribute addProperty Name "R6 (EK1100)"}
TYPE R6_EK1100_8C41F5F2 EXTENDS EK1100_1FC0878B :
STRUCT
    {attribute addProperty Name "R6_A2_DI (EL1809)"}
    {attribute addProperty PreviousPort "R6 (EK1100) : B"}
    {attribute addProperty SyncUnit "default"}
    R6_A2_DI_EL1809 : EL1809_32157CFD;
    {attribute addProperty Name "R6_A3_DI (EL1809)"}
    {attribute addProperty PreviousPort "R6_A2_DI (EL1809) : B"}
    {attribute addProperty SyncUnit "default"}
    R6_A3_DI_EL1809 : EL1809_32157CFD;
    {attribute addProperty Name "R6_A4_DI (EL1809)"}
    {attribute addProperty PreviousPort "R6_A3_DI (EL1809) : B"}
    {attribute addProperty SyncUnit "default"}
    R6_A4_DI_EL1809 : EL1809_32157CFD;
    {attribute addProperty Name "R6_A5_DI (EL1809)"}
    {attribute addProperty PreviousPort "R6_A4_DI (EL1809) : B"}
    {attribute addProperty SyncUnit "default"}
    R6_A5_DI_EL1809 : EL1809_32157CFD;
    {attribute addProperty Name "R6_A6_DI (EL1809)"}
    {attribute addProperty PreviousPort "R6_A5_DI (EL1809) : B"}
    {attribute addProperty SyncUnit "default"}
    R6_A6_DI_EL1809 : EL1809_32157CFD;
    {attribute addProperty Name "R6_A7_DI (EL1809)"}
    {attribute addProperty PreviousPort "R6_A6_DI (EL1809) : B"}
    {attribute addProperty SyncUnit "default"}
    R6_A7_DI_EL1809 : EL1809_32157CFD;
    {attribute addProperty Name "R6_A8_DI (EL1809)"}
    {attribute addProperty PreviousPort "R6_A7_DI (EL1809) : B"}
    {attribute addProperty SyncUnit "default"}
    R6_A8_DI_EL1809 : EL1809_32157CFD;
    {attribute addProperty Name "R6_A9_DI (EL1809)"}
    {attribute addProperty PreviousPort "R6_A8_DI (EL1809) : B"}
    {attribute addProperty SyncUnit "default"}
    R6_A9_DI_EL1809 : EL1809_32157CFD;
    {attribute addProperty Name "R6_A10_DI (EL1809)"}
    {attribute addProperty PreviousPort "R6_A9_DI (EL1809) : B"}
    {attribute addProperty SyncUnit "default"}
    R6_A10_DI_EL1809 : EL1809_32157CFD;
    {attribute addProperty Name "R6_A11_DI (EL1809)"}
    {attribute addProperty PreviousPort "R6_A10_DI (EL1809) : B"}
    {attribute addProperty SyncUnit "default"}
    R6_A11_DI_EL1809 : EL1809_32157CFD;
    {attribute addProperty Name "R6_A12_DI (EL1809)"}
    {attribute addProperty PreviousPort "R6_A11_DI (EL1809) : B"}
    {attribute addProperty SyncUnit "default"}
    R6_A12_DI_EL1809 : EL1809_32157CFD;
    {attribute addProperty Name "R6_A13_DI (EL1809)"}
    {attribute addProperty PreviousPort "R6_A12_DI (EL1809) : B"}
    {attribute addProperty SyncUnit "default"}
    R6_A13_DI_EL1809 : EL1809_32157CFD;
    {attribute addProperty Name "R6_A14_DI (EL1809)"}
    {attribute addProperty PreviousPort "R6_A13_DI (EL1809) : B"}
    {attribute addProperty SyncUnit "default"}
    R6_A14_DI_EL1809 : EL1809_32157CFD;
    {attribute addProperty Name "R6_A15_DO (EL2809)"}
    {attribute addProperty PreviousPort "R6_A14_DI (EL1809) : B"}
    {attribute addProperty SyncUnit "default"}
    R6_A15_DO_EL2809 : EL2809_2B6483BD;
    {attribute addProperty Name "R6_A16_DO (EL2809)"}
    {attribute addProperty PreviousPort "R6_A15_DO (EL2809) : B"}
    {attribute addProperty SyncUnit "default"}
    R6_A16_DO_EL2809 : EL2809_2B6483BD;
    {attribute addProperty Name "R6_A17_DO (EL2809)"}
    {attribute addProperty PreviousPort "R6_A16_DO (EL2809) : B"}
    {attribute addProperty SyncUnit "default"}
    R6_A17_DO_EL2809 : EL2809_2B6483BD;
    {attribute addProperty Name "R6_A18_DO (EL2809)"}
    {attribute addProperty PreviousPort "R6_A17_DO (EL2809) : B"}
    {attribute addProperty SyncUnit "default"}
    R6_A18_DO_EL2809 : EL2809_2B6483BD;
    {attribute addProperty Name "R6_EndTerminal (EL9011)"}
    {attribute addProperty PreviousPort "R6_A18_DO (EL2809) : B"}
    {attribute addProperty SyncUnit "default"}
    R6_EndTerminal_EL9011 : EL9011_D65D3D32;
END_STRUCT
END_TYPE

// ---- DUTs/IO/Topology/R7_A2_EC_EK1122_B7F046E4.TcDUT
{attribute 'GeneratedUsingTerminal: EK1122-0000-0018'}
{attribute addProperty BoxType "EK1122-0000-0018"}
{attribute addProperty Id "VI_6_AES_D_BC_ECAT_xAES_A3B0707168"}
{attribute addProperty CRC "3085977316"}
{attribute addProperty Size "68"}
{attribute addProperty Name "R7_A2_EC (EK1122)"}
TYPE R7_A2_EC_EK1122_B7F046E4 EXTENDS EK1122_1FC0878B :
STRUCT
    {attribute addProperty Name "VI-6 (AES-D-BC-ECAT)"}
    {attribute addProperty PreviousPort "R7_A2_EC (EK1122) : D"}
    {attribute addProperty SyncUnit "default"}
    VI_6_AES_D_BC_ECAT_x : AES_A3B07071;
END_STRUCT
END_TYPE

// ---- DUTs/IO/Topology/R7_EK1100_F50DDAC8.TcDUT
{attribute 'GeneratedUsingTerminal: EK1100-0000-0018'}
{attribute addProperty BoxType "EK1100-0000-0018"}
{attribute addProperty Id "R7_A2_EC_EK1122R7_A2_EC_EK1122_B7F046E468R7_A3_DI_EL1809EL1809_32157CFD20R7_A4_DI_EL1809EL1809_32157CFD20R7_A5_DI_EL1809EL1809_32157CFD20R7_A6_DI_EL1809EL1809_32157CFD20R7_A7_DI_EL1809EL1809_32157CFD20R7_A8_DI_EL1809EL1809_32157CFD20R7_A9_DI_EL1809EL1809_32157CFD20R7_A10_DI_EL1809EL1809_32157CFD20R7_A11_DI_EL1809EL1809_32157CFD20R7_A12_DI_EL1809EL1809_32157CFD20R7_A13_DI_EL2809EL2809_2B6483BD19R7_A14_DI_EL2809EL2809_2B6483BD19R7_EndTerminal_EL9011EL9011_D65D3D320"}
{attribute addProperty CRC "4111325896"}
{attribute addProperty Size "306"}
{attribute addProperty Name "R7 (EK1100)"}
TYPE R7_EK1100_F50DDAC8 EXTENDS EK1100_1FC0878B :
STRUCT
    {attribute addProperty Name "R7_A2_EC (EK1122)"}
    {attribute addProperty PreviousPort "R7 (EK1100) : B"}
    {attribute addProperty SyncUnit "default"}
    R7_A2_EC_EK1122 : R7_A2_EC_EK1122_B7F046E4;
    {attribute addProperty Name "R7_A3_DI (EL1809)"}
    {attribute addProperty PreviousPort "R7_A2_EC (EK1122) : C"}
    {attribute addProperty SyncUnit "default"}
    R7_A3_DI_EL1809 : EL1809_32157CFD;
    {attribute addProperty Name "R7_A4_DI (EL1809)"}
    {attribute addProperty PreviousPort "R7_A3_DI (EL1809) : B"}
    {attribute addProperty SyncUnit "default"}
    R7_A4_DI_EL1809 : EL1809_32157CFD;
    {attribute addProperty Name "R7_A5_DI (EL1809)"}
    {attribute addProperty PreviousPort "R7_A4_DI (EL1809) : B"}
    {attribute addProperty SyncUnit "default"}
    R7_A5_DI_EL1809 : EL1809_32157CFD;
    {attribute addProperty Name "R7_A6_DI (EL1809)"}
    {attribute addProperty PreviousPort "R7_A5_DI (EL1809) : B"}
    {attribute addProperty SyncUnit "default"}
    R7_A6_DI_EL1809 : EL1809_32157CFD;
    {attribute addProperty Name "R7_A7_DI (EL1809)"}
    {attribute addProperty PreviousPort "R7_A6_DI (EL1809) : B"}
    {attribute addProperty SyncUnit "default"}
    R7_A7_DI_EL1809 : EL1809_32157CFD;
    {attribute addProperty Name "R7_A8_DI (EL1809)"}
    {attribute addProperty PreviousPort "R7_A7_DI (EL1809) : B"}
    {attribute addProperty SyncUnit "default"}
    R7_A8_DI_EL1809 : EL1809_32157CFD;
    {attribute addProperty Name "R7_A9_DI (EL1809)"}
    {attribute addProperty PreviousPort "R7_A8_DI (EL1809) : B"}
    {attribute addProperty SyncUnit "default"}
    R7_A9_DI_EL1809 : EL1809_32157CFD;
    {attribute addProperty Name "R7_A10_DI (EL1809)"}
    {attribute addProperty PreviousPort "R7_A9_DI (EL1809) : B"}
    {attribute addProperty SyncUnit "default"}
    R7_A10_DI_EL1809 : EL1809_32157CFD;
    {attribute addProperty Name "R7_A11_DI (EL1809)"}
    {attribute addProperty PreviousPort "R7_A10_DI (EL1809) : B"}
    {attribute addProperty SyncUnit "default"}
    R7_A11_DI_EL1809 : EL1809_32157CFD;
    {attribute addProperty Name "R7_A12_DI (EL1809)"}
    {attribute addProperty PreviousPort "R7_A11_DI (EL1809) : B"}
    {attribute addProperty SyncUnit "default"}
    R7_A12_DI_EL1809 : EL1809_32157CFD;
    {attribute addProperty Name "R7_A13_DI (EL2809)"}
    {attribute addProperty PreviousPort "R7_A12_DI (EL1809) : B"}
    {attribute addProperty SyncUnit "default"}
    R7_A13_DI_EL2809 : EL2809_2B6483BD;
    {attribute addProperty Name "R7_A14_DI (EL2809)"}
    {attribute addProperty PreviousPort "R7_A13_DI (EL2809) : B"}
    {attribute addProperty SyncUnit "default"}
    R7_A14_DI_EL2809 : EL2809_2B6483BD;
    {attribute addProperty Name "R7_EndTerminal (EL9011)"}
    {attribute addProperty PreviousPort "R7_A14_DI (EL2809) : B"}
    {attribute addProperty SyncUnit "default"}
    R7_EndTerminal_EL9011 : EL9011_D65D3D32;
END_STRUCT
END_TYPE

// ---- DUTs/IO/Topology/R8_AB0_EPP1322_0001_1BB6BCA8.TcDUT
{attribute 'GeneratedUsingTerminal: EPP1322-0001-0017'}
{attribute addProperty BoxType "EPP1322-0001-0017"}
{attribute addProperty Id "R8_AB24_EPP1008_0001EPP1008_78E8D3DD12R8_AB23_EPP1008_0001EPP1008_78E8D3DD12R8_AB22_EPP1008_0001EPP1008_78E8D3DD12R8_AB21_EPP1008_0001EPP1008_78E8D3DD12R8_AB20_EPP1008_0001EPP1008_78E8D3DD12R8_AB19_EPP1008_0001EPP1008_78E8D3DD12R8_AB18_EPP1008_0001EPP1008_78E8D3DD12R8_AB17_EPP1008_0001EPP1008_78E8D3DD12R8_AB16_EPP1008_0001EPP1008_78E8D3DD12R8_AB15_EPP1008_0001EPP1008_78E8D3DD12R8_AB14_EPP1008_0001EPP1008_78E8D3DD12R8_AB13_EPP1008_0001EPP1008_78E8D3DD12Box_379_EPP1332_0001EPP1332_1FC0878B2R8_AB12_EPP1008_0001EPP1008_78E8D3DD12R8_AB11_EPP1008_0001EPP1008_78E8D3DD12R8_AB10_EPP1008_0001EPP1008_78E8D3DD12R8_AB9_EPP1008_0001EPP1008_78E8D3DD12R8_AB8_EPP1008_0001EPP1008_78E8D3DD12R8_AB7_EPP1008_0001EPP1008_78E8D3DD12R8_AB6_EPP1008_0001EPP1008_78E8D3DD12R8_AB5_EPP1008_0001EPP1008_78E8D3DD12R8_AB4_EPP1008_0001EPP1008_78E8D3DD12R8_AB3_EPP1008_0001EPP1008_78E8D3DD12R8_AB2_EPP1008_0001EPP1008_78E8D3DD12R8_AB1_EPP1008_0001EPP1008_78E8D3DD12"}
{attribute addProperty CRC "464960680"}
{attribute addProperty Size "290"}
{attribute addProperty Name "R8_AB0 (EPP1322-0001)"}
TYPE R8_AB0_EPP1322_0001_1BB6BCA8 EXTENDS EPP1322_1FC0878B :
STRUCT
    {attribute addProperty Name "R8_AB24 (EPP1008-0001)"}
    {attribute addProperty PreviousPort "R8_AB0 (EPP1322-0001) : D"}
    {attribute addProperty SyncUnit "default"}
    R8_AB24_EPP1008_0001 : EPP1008_78E8D3DD;
    {attribute addProperty Name "R8_AB23 (EPP1008-0001)"}
    {attribute addProperty PreviousPort "R8_AB24 (EPP1008-0001) : B"}
    {attribute addProperty SyncUnit "default"}
    R8_AB23_EPP1008_0001 : EPP1008_78E8D3DD;
    {attribute addProperty Name "R8_AB22 (EPP1008-0001)"}
    {attribute addProperty PreviousPort "R8_AB23 (EPP1008-0001) : B"}
    {attribute addProperty SyncUnit "default"}
    R8_AB22_EPP1008_0001 : EPP1008_78E8D3DD;
    {attribute addProperty Name "R8_AB21 (EPP1008-0001)"}
    {attribute addProperty PreviousPort "R8_AB22 (EPP1008-0001) : B"}
    {attribute addProperty SyncUnit "default"}
    R8_AB21_EPP1008_0001 : EPP1008_78E8D3DD;
    {attribute addProperty Name "R8_AB20 (EPP1008-0001)"}
    {attribute addProperty PreviousPort "R8_AB21 (EPP1008-0001) : B"}
    {attribute addProperty SyncUnit "default"}
    R8_AB20_EPP1008_0001 : EPP1008_78E8D3DD;
    {attribute addProperty Name "R8_AB19 (EPP1008-0001)"}
    {attribute addProperty PreviousPort "R8_AB20 (EPP1008-0001) : B"}
    {attribute addProperty SyncUnit "default"}
    R8_AB19_EPP1008_0001 : EPP1008_78E8D3DD;
    {attribute addProperty Name "R8_AB18 (EPP1008-0001)"}
    {attribute addProperty PreviousPort "R8_AB19 (EPP1008-0001) : B"}
    {attribute addProperty SyncUnit "default"}
    R8_AB18_EPP1008_0001 : EPP1008_78E8D3DD;
    {attribute addProperty Name "R8_AB17 (EPP1008-0001)"}
    {attribute addProperty PreviousPort "R8_AB18 (EPP1008-0001) : B"}
    {attribute addProperty SyncUnit "default"}
    R8_AB17_EPP1008_0001 : EPP1008_78E8D3DD;
    {attribute addProperty Name "R8_AB16 (EPP1008-0001)"}
    {attribute addProperty PreviousPort "R8_AB17 (EPP1008-0001) : B"}
    {attribute addProperty SyncUnit "default"}
    R8_AB16_EPP1008_0001 : EPP1008_78E8D3DD;
    {attribute addProperty Name "R8_AB15 (EPP1008-0001)"}
    {attribute addProperty PreviousPort "R8_AB16 (EPP1008-0001) : B"}
    {attribute addProperty SyncUnit "default"}
    R8_AB15_EPP1008_0001 : EPP1008_78E8D3DD;
    {attribute addProperty Name "R8_AB14 (EPP1008-0001)"}
    {attribute addProperty PreviousPort "R8_AB15 (EPP1008-0001) : B"}
    {attribute addProperty SyncUnit "default"}
    R8_AB14_EPP1008_0001 : EPP1008_78E8D3DD;
    {attribute addProperty Name "R8_AB13 (EPP1008-0001)"}
    {attribute addProperty PreviousPort "R8_AB14 (EPP1008-0001) : B"}
    {attribute addProperty SyncUnit "default"}
    R8_AB13_EPP1008_0001 : EPP1008_78E8D3DD;
    {attribute addProperty Name "Box 379 (EPP1332-0001)"}
    {attribute addProperty PreviousPort "R8_AB13 (EPP1008-0001) : B"}
    {attribute addProperty SyncUnit "default"}
    Box_379_EPP1332_0001 : EPP1332_1FC0878B;
    {attribute addProperty Name "R8_AB12 (EPP1008-0001)"}
    {attribute addProperty PreviousPort "Box 379 (EPP1332-0001) : C"}
    {attribute addProperty SyncUnit "default"}
    R8_AB12_EPP1008_0001 : EPP1008_78E8D3DD;
    {attribute addProperty Name "R8_AB11 (EPP1008-0001)"}
    {attribute addProperty PreviousPort "R8_AB12 (EPP1008-0001) : B"}
    {attribute addProperty SyncUnit "default"}
    R8_AB11_EPP1008_0001 : EPP1008_78E8D3DD;
    {attribute addProperty Name "R8_AB10 (EPP1008-0001)"}
    {attribute addProperty PreviousPort "R8_AB11 (EPP1008-0001) : B"}
    {attribute addProperty SyncUnit "default"}
    R8_AB10_EPP1008_0001 : EPP1008_78E8D3DD;
    {attribute addProperty Name "R8_AB9 (EPP1008-0001)"}
    {attribute addProperty PreviousPort "R8_AB10 (EPP1008-0001) : B"}
    {attribute addProperty SyncUnit "default"}
    R8_AB9_EPP1008_0001 : EPP1008_78E8D3DD;
    {attribute addProperty Name "R8_AB8 (EPP1008-0001)"}
    {attribute addProperty PreviousPort "R8_AB9 (EPP1008-0001) : B"}
    {attribute addProperty SyncUnit "default"}
    R8_AB8_EPP1008_0001 : EPP1008_78E8D3DD;
    {attribute addProperty Name "R8_AB7 (EPP1008-0001)"}
    {attribute addProperty PreviousPort "R8_AB8 (EPP1008-0001) : B"}
    {attribute addProperty SyncUnit "default"}
    R8_AB7_EPP1008_0001 : EPP1008_78E8D3DD;
    {attribute addProperty Name "R8_AB6 (EPP1008-0001)"}
    {attribute addProperty PreviousPort "R8_AB7 (EPP1008-0001) : B"}
    {attribute addProperty SyncUnit "default"}
    R8_AB6_EPP1008_0001 : EPP1008_78E8D3DD;
    {attribute addProperty Name "R8_AB5 (EPP1008-0001)"}
    {attribute addProperty PreviousPort "R8_AB6 (EPP1008-0001) : B"}
    {attribute addProperty SyncUnit "default"}
    R8_AB5_EPP1008_0001 : EPP1008_78E8D3DD;
    {attribute addProperty Name "R8_AB4 (EPP1008-0001)"}
    {attribute addProperty PreviousPort "R8_AB5 (EPP1008-0001) : B"}
    {attribute addProperty SyncUnit "default"}
    R8_AB4_EPP1008_0001 : EPP1008_78E8D3DD;
    {attribute addProperty Name "R8_AB3 (EPP1008-0001)"}
    {attribute addProperty PreviousPort "R8_AB4 (EPP1008-0001) : B"}
    {attribute addProperty SyncUnit "default"}
    R8_AB3_EPP1008_0001 : EPP1008_78E8D3DD;
    {attribute addProperty Name "R8_AB2 (EPP1008-0001)"}
    {attribute addProperty PreviousPort "R8_AB3 (EPP1008-0001) : B"}
    {attribute addProperty SyncUnit "default"}
    R8_AB2_EPP1008_0001 : EPP1008_78E8D3DD;
    {attribute addProperty Name "R8_AB1 (EPP1008-0001)"}
    {attribute addProperty PreviousPort "R8_AB2 (EPP1008-0001) : B"}
    {attribute addProperty SyncUnit "default"}
    R8_AB1_EPP1008_0001 : EPP1008_78E8D3DD;
END_STRUCT
END_TYPE

// ---- DUTs/IO/Topology/R8_A2_EK1122_E74C4B62.TcDUT
{attribute 'GeneratedUsingTerminal: EK1122-0000-0018'}
{attribute addProperty BoxType "EK1122-0000-0018"}
{attribute addProperty Id "R8_AB0_EPP1322_0001R8_AB0_EPP1322_0001_1BB6BCA8290"}
{attribute addProperty CRC "3880536930"}
{attribute addProperty Size "290"}
{attribute addProperty Name "R8_A2 (EK1122)"}
TYPE R8_A2_EK1122_E74C4B62 EXTENDS EK1122_1FC0878B :
STRUCT
    {attribute addProperty Name "R8_AB0 (EPP1322-0001)"}
    {attribute addProperty PreviousPort "R8_A2 (EK1122) : D"}
    {attribute addProperty SyncUnit "default"}
    R8_AB0_EPP1322_0001 : R8_AB0_EPP1322_0001_1BB6BCA8;
END_STRUCT
END_TYPE

// ---- DUTs/IO/Topology/R8_A3_EK1122_71CA94BA.TcDUT
{attribute 'GeneratedUsingTerminal: EK1122-0000-0018'}
{attribute addProperty BoxType "EK1122-0000-0018"}
{attribute addProperty Id "VI_10_AES_D_BC_ECAT_xAES_A3B0707168VI_9_AES_D_BC_ECAT_xAES_A3B0707168"}
{attribute addProperty CRC "1909101754"}
{attribute addProperty Size "136"}
{attribute addProperty Name "R8_A3 (EK1122)"}
TYPE R8_A3_EK1122_71CA94BA EXTENDS EK1122_1FC0878B :
STRUCT
    {attribute addProperty Name "VI-10 (AES-D-BC-ECAT)"}
    {attribute addProperty PreviousPort "R8_A3 (EK1122) : D"}
    {attribute addProperty SyncUnit "default"}
    VI_10_AES_D_BC_ECAT_x : AES_A3B07071;
    {attribute addProperty Name "VI-9 (AES-D-BC-ECAT)"}
    {attribute addProperty PreviousPort "R8_A3 (EK1122) : B"}
    {attribute addProperty SyncUnit "default"}
    VI_9_AES_D_BC_ECAT_x : AES_A3B07071;
END_STRUCT
END_TYPE

// ---- DUTs/IO/Topology/RC10_A2_EK1122_BBB6F36B.TcDUT
{attribute 'GeneratedUsingTerminal: EK1122-0000-0018'}
{attribute addProperty BoxType "EK1122-0000-0018"}
{attribute addProperty Id "RC10_VI_AES_D_BC_ECAT_xAES_A3B0707168RC10_SAFETY_Flexi_Soft_EtherCAT_GatewayFlexi_Soft_EtherCAT_Gateway_DE394EDD5"}
{attribute addProperty CRC "3149329259"}
{attribute addProperty Size "73"}
{attribute addProperty Name "RC10_A2 (EK1122)"}
TYPE RC10_A2_EK1122_BBB6F36B EXTENDS EK1122_1FC0878B :
STRUCT
    {attribute addProperty Name "RC10_VI (AES-D-BC-ECAT)"}
    {attribute addProperty PreviousPort "RC10_A2 (EK1122) : D"}
    {attribute addProperty SyncUnit "C10"}
    RC10_VI_AES_D_BC_ECAT_x : AES_A3B07071;
    {attribute addProperty Name "RC10_SAFETY (Flexi Soft EtherCAT Gateway)"}
    {attribute addProperty PreviousPort "RC10_A2 (EK1122) : B"}
    {attribute addProperty SyncUnit "C10"}
    RC10_SAFETY_Flexi_Soft_EtherCAT_Gateway : Flexi_Soft_EtherCAT_Gateway_DE394EDD;
END_STRUCT
END_TYPE

// ---- DUTs/IO/Topology/RC10_EPP_EPP1322_0001_810E0540.TcDUT
{attribute 'GeneratedUsingTerminal: EPP1322-0001-0017'}
{attribute addProperty BoxType "EPP1322-0001-0017"}
{attribute addProperty Id "RC10_AB1_EPP1008_0001EPP1008_78E8D3DD12RC10_AB2_EPP1008_0001EPP1008_78E8D3DD12RC10_AB6_EPP1008_0001EPP1008_78E8D3DD12RC10_AB3_EPP1008_0001EPP1008_78E8D3DD12RC10_AB4_EPP1008_0001EPP1008_78E8D3DD12RC10_AB7_EPP1008_0001EPP1008_78E8D3DD12RC10_AB9_EPP1008_0001EPP1008_78E8D3DD12RC10_AB10_EPP1008_0001EPP1008_78E8D3DD12RC10_AB8_EPP1008_0001EPP1008_78E8D3DD12RC10_AB5_EPP1008_0001EPP1008_78E8D3DD12"}
{attribute addProperty CRC "2165179712"}
{attribute addProperty Size "120"}
{attribute addProperty Name "RC10_EPP (EPP1322-0001)"}
TYPE RC10_EPP_EPP1322_0001_810E0540 EXTENDS EPP1322_1FC0878B :
STRUCT
    {attribute addProperty Name "RC10_AB1 (EPP1008-0001)"}
    {attribute addProperty PreviousPort "RC10_EPP (EPP1322-0001) : D"}
    {attribute addProperty SyncUnit "C10"}
    RC10_AB1_EPP1008_0001 : EPP1008_78E8D3DD;
    {attribute addProperty Name "RC10_AB2 (EPP1008-0001)"}
    {attribute addProperty PreviousPort "RC10_AB1 (EPP1008-0001) : B"}
    {attribute addProperty SyncUnit "C10"}
    RC10_AB2_EPP1008_0001 : EPP1008_78E8D3DD;
    {attribute addProperty Name "RC10_AB6 (EPP1008-0001)"}
    {attribute addProperty PreviousPort "RC10_AB2 (EPP1008-0001) : B"}
    {attribute addProperty SyncUnit "C10"}
    RC10_AB6_EPP1008_0001 : EPP1008_78E8D3DD;
    {attribute addProperty Name "RC10_AB3 (EPP1008-0001)"}
    {attribute addProperty PreviousPort "RC10_AB6 (EPP1008-0001) : B"}
    {attribute addProperty SyncUnit "C10"}
    RC10_AB3_EPP1008_0001 : EPP1008_78E8D3DD;
    {attribute addProperty Name "RC10_AB4 (EPP1008-0001)"}
    {attribute addProperty PreviousPort "RC10_AB3 (EPP1008-0001) : B"}
    {attribute addProperty SyncUnit "C10"}
    RC10_AB4_EPP1008_0001 : EPP1008_78E8D3DD;
    {attribute addProperty Name "RC10_AB7 (EPP1008-0001)"}
    {attribute addProperty PreviousPort "RC10_EPP (EPP1322-0001) : B"}
    {attribute addProperty SyncUnit "C10"}
    RC10_AB7_EPP1008_0001 : EPP1008_78E8D3DD;
    {attribute addProperty Name "RC10_AB9 (EPP1008-0001)"}
    {attribute addProperty PreviousPort "RC10_AB7 (EPP1008-0001) : B"}
    {attribute addProperty SyncUnit "C10"}
    RC10_AB9_EPP1008_0001 : EPP1008_78E8D3DD;
    {attribute addProperty Name "RC10_AB10 (EPP1008-0001)"}
    {attribute addProperty PreviousPort "RC10_AB9 (EPP1008-0001) : B"}
    {attribute addProperty SyncUnit "C10"}
    RC10_AB10_EPP1008_0001 : EPP1008_78E8D3DD;
    {attribute addProperty Name "RC10_AB8 (EPP1008-0001)"}
    {attribute addProperty PreviousPort "RC10_AB10 (EPP1008-0001) : B"}
    {attribute addProperty SyncUnit "C10"}
    RC10_AB8_EPP1008_0001 : EPP1008_78E8D3DD;
    {attribute addProperty Name "RC10_AB5 (EPP1008-0001)"}
    {attribute addProperty PreviousPort "RC10_AB8 (EPP1008-0001) : B"}
    {attribute addProperty SyncUnit "C10"}
    RC10_AB5_EPP1008_0001 : EPP1008_78E8D3DD;
END_STRUCT
END_TYPE

// ---- DUTs/IO/Topology/RC10_A3_EK1122_A50FC1ED.TcDUT
{attribute 'GeneratedUsingTerminal: EK1122-0000-0018'}
{attribute addProperty BoxType "EK1122-0000-0018"}
{attribute addProperty Id "RC10_EPP_EPP1322_0001RC10_EPP_EPP1322_0001_810E0540120"}
{attribute addProperty CRC "2769273325"}
{attribute addProperty Size "120"}
{attribute addProperty Name "RC10_A3 (EK1122)"}
TYPE RC10_A3_EK1122_A50FC1ED EXTENDS EK1122_1FC0878B :
STRUCT
    {attribute addProperty Name "RC10_EPP (EPP1322-0001)"}
    {attribute addProperty PreviousPort "RC10_A3 (EK1122) : D"}
    {attribute addProperty SyncUnit "default"}
    RC10_EPP_EPP1322_0001 : RC10_EPP_EPP1322_0001_810E0540;
END_STRUCT
END_TYPE

// ---- DUTs/IO/Topology/RC10_1_EK1100_40BAEC0F.TcDUT
{attribute 'GeneratedUsingTerminal: EK1100-0000-0018'}
{attribute addProperty BoxType "EK1100-0000-0018"}
{attribute addProperty Id "RC10_A2_EK1122RC10_A2_EK1122_BBB6F36B73RC10_A3_EK1122RC10_A3_EK1122_A50FC1ED120RC10_A5_EL1809EL1809_32157CFD20RC10_A6_EL1809EL1809_32157CFD20RC10_A7_EL2809EL2809_2B6483BD19RC10_A8_EL2809EL2809_2B6483BD19RC10_A9_EL2809EL2809_2B6483BD19RC10_1_EndTerminal_EL9011EL9011_D65D3D320"}
{attribute addProperty CRC "1085991951"}
{attribute addProperty Size "290"}
{attribute addProperty Name "RC10_1 (EK1100)"}
TYPE RC10_1_EK1100_40BAEC0F EXTENDS EK1100_1FC0878B :
STRUCT
    {attribute addProperty Name "RC10_A2 (EK1122)"}
    {attribute addProperty PreviousPort "RC10_1 (EK1100) : B"}
    {attribute addProperty SyncUnit "default"}
    RC10_A2_EK1122 : RC10_A2_EK1122_BBB6F36B;
    {attribute addProperty Name "RC10_A3 (EK1122)"}
    {attribute addProperty PreviousPort "RC10_A2 (EK1122) : C"}
    {attribute addProperty SyncUnit "default"}
    RC10_A3_EK1122 : RC10_A3_EK1122_A50FC1ED;
    {attribute addProperty Name "RC10_A5 (EL1809)"}
    {attribute addProperty PreviousPort "RC10_A3 (EK1122) : C"}
    {attribute addProperty SyncUnit "C10"}
    RC10_A5_EL1809 : EL1809_32157CFD;
    {attribute addProperty Name "RC10_A6 (EL1809)"}
    {attribute addProperty PreviousPort "RC10_A5 (EL1809) : B"}
    {attribute addProperty SyncUnit "C10"}
    RC10_A6_EL1809 : EL1809_32157CFD;
    {attribute addProperty Name "RC10_A7 (EL2809)"}
    {attribute addProperty PreviousPort "RC10_A6 (EL1809) : B"}
    {attribute addProperty SyncUnit "C10"}
    RC10_A7_EL2809 : EL2809_2B6483BD;
    {attribute addProperty Name "RC10_A8 (EL2809)"}
    {attribute addProperty PreviousPort "RC10_A7 (EL2809) : B"}
    {attribute addProperty SyncUnit "C10"}
    RC10_A8_EL2809 : EL2809_2B6483BD;
    {attribute addProperty Name "RC10_A9 (EL2809)"}
    {attribute addProperty PreviousPort "RC10_A8 (EL2809) : B"}
    {attribute addProperty SyncUnit "C10"}
    RC10_A9_EL2809 : EL2809_2B6483BD;
    {attribute addProperty Name "RC10_1_EndTerminal (EL9011)"}
    {attribute addProperty PreviousPort "RC10_A9 (EL2809) : B"}
    {attribute addProperty SyncUnit "default"}
    RC10_1_EndTerminal_EL9011 : EL9011_D65D3D32;
END_STRUCT
END_TYPE

// ---- DUTs/IO/Topology/RC10_2_EK1100_27865421.TcDUT
{attribute 'GeneratedUsingTerminal: EK1100-0000-0018'}
{attribute addProperty BoxType "EK1100-0000-0018"}
{attribute addProperty Id "RC10_B1_EL7041_1000EL7041_86DE63E743RC10_B2_EL7041_1000EL7041_86DE63E743RC10_C11_EL7041_1000EL7041_86DE63E743RC10_C12_EL7041_1000EL7041_86DE63E743RC10_C21_EL7041_1000EL7041_86DE63E743RC10_C22_EL7041_1000EL7041_86DE63E743RC10_2_EndTerminal_EL9010EL9010_D29C20850"}
{attribute addProperty CRC "663114785"}
{attribute addProperty Size "258"}
{attribute addProperty Name "RC10_2 (EK1100)"}
TYPE RC10_2_EK1100_27865421 EXTENDS EK1100_1FC0878B :
STRUCT
    {attribute addProperty Name "RC10_B1 (EL7041-1000)"}
    {attribute addProperty PreviousPort "RC10_2 (EK1100) : B"}
    {attribute addProperty SyncUnit "C10"}
    RC10_B1_EL7041_1000 : EL7041_86DE63E7;
    {attribute addProperty Name "RC10_B2 (EL7041-1000)"}
    {attribute addProperty PreviousPort "RC10_B1 (EL7041-1000) : B"}
    {attribute addProperty SyncUnit "C10"}
    RC10_B2_EL7041_1000 : EL7041_86DE63E7;
    {attribute addProperty Name "RC10_C11 (EL7041-1000)"}
    {attribute addProperty PreviousPort "RC10_B2 (EL7041-1000) : B"}
    {attribute addProperty SyncUnit "C10"}
    RC10_C11_EL7041_1000 : EL7041_86DE63E7;
    {attribute addProperty Name "RC10_C12 (EL7041-1000)"}
    {attribute addProperty PreviousPort "RC10_C11 (EL7041-1000) : B"}
    {attribute addProperty SyncUnit "C10"}
    RC10_C12_EL7041_1000 : EL7041_86DE63E7;
    {attribute addProperty Name "RC10_C21 (EL7041-1000)"}
    {attribute addProperty PreviousPort "RC10_C12 (EL7041-1000) : B"}
    {attribute addProperty SyncUnit "C10"}
    RC10_C21_EL7041_1000 : EL7041_86DE63E7;
    {attribute addProperty Name "RC10_C22 (EL7041-1000)"}
    {attribute addProperty PreviousPort "RC10_C21 (EL7041-1000) : B"}
    {attribute addProperty SyncUnit "C10"}
    RC10_C22_EL7041_1000 : EL7041_86DE63E7;
    {attribute addProperty Name "RC10_2_EndTerminal (EL9010)"}
    {attribute addProperty PreviousPort "RC10_C22 (EL7041-1000) : B"}
    {attribute addProperty SyncUnit "default"}
    RC10_2_EndTerminal_EL9010 : EL9010_D29C2085;
END_STRUCT
END_TYPE

// ---- DUTs/IO/Topology/RC20_A2_EK1122_77321D67.TcDUT
{attribute 'GeneratedUsingTerminal: EK1122-0000-0018'}
{attribute addProperty BoxType "EK1122-0000-0018"}
{attribute addProperty Id "RC20_VI_AES_D_BC_ECAT_xAES_A3B0707168RC20_SAFETY_Flexi_Soft_EtherCAT_GatewayFlexi_Soft_EtherCAT_Gateway_DE394EDD5"}
{attribute addProperty CRC "1999773031"}
{attribute addProperty Size "73"}
{attribute addProperty Name "RC20_A2 (EK1122)"}
TYPE RC20_A2_EK1122_77321D67 EXTENDS EK1122_1FC0878B :
STRUCT
    {attribute addProperty Name "RC20_VI (AES-D-BC-ECAT)"}
    {attribute addProperty PreviousPort "RC20_A2 (EK1122) : D"}
    {attribute addProperty SyncUnit "C20"}
    RC20_VI_AES_D_BC_ECAT_x : AES_A3B07071;
    {attribute addProperty Name "RC20_SAFETY (Flexi Soft EtherCAT Gateway)"}
    {attribute addProperty PreviousPort "RC20_A2 (EK1122) : B"}
    {attribute addProperty SyncUnit "C20"}
    RC20_SAFETY_Flexi_Soft_EtherCAT_Gateway : Flexi_Soft_EtherCAT_Gateway_DE394EDD;
END_STRUCT
END_TYPE

// ---- DUTs/IO/Topology/RC20_EPP_EPP1322_0001_59D450BA.TcDUT
{attribute 'GeneratedUsingTerminal: EPP1322-0001-0017'}
{attribute addProperty BoxType "EPP1322-0001-0017"}
{attribute addProperty Id "RC20_AB1_EPP1008_0001EPP1008_78E8D3DD12RC20_AB2_EPP1008_0001EPP1008_78E8D3DD12RC20_AB6_EPP1008_0001EPP1008_78E8D3DD12RC20_AB3_EPP1008_0001EPP1008_78E8D3DD12RC20_AB4_EPP1008_0001EPP1008_78E8D3DD12RC20_AB7_EPP1008_0001EPP1008_78E8D3DD12RC20_AB9_EPP1008_0001EPP1008_78E8D3DD12RC20_AB10_EPP1008_0001EPP1008_78E8D3DD12RC20_AB8_EPP1008_0001EPP1008_78E8D3DD12RC20_AB5_EPP1008_0001EPP1008_78E8D3DD12"}
{attribute addProperty CRC "1507086522"}
{attribute addProperty Size "120"}
{attribute addProperty Name "RC20_EPP (EPP1322-0001)"}
TYPE RC20_EPP_EPP1322_0001_59D450BA EXTENDS EPP1322_1FC0878B :
STRUCT
    {attribute addProperty Name "RC20_AB1 (EPP1008-0001)"}
    {attribute addProperty PreviousPort "RC20_EPP (EPP1322-0001) : D"}
    {attribute addProperty SyncUnit "C20"}
    RC20_AB1_EPP1008_0001 : EPP1008_78E8D3DD;
    {attribute addProperty Name "RC20_AB2 (EPP1008-0001)"}
    {attribute addProperty PreviousPort "RC20_AB1 (EPP1008-0001) : B"}
    {attribute addProperty SyncUnit "C20"}
    RC20_AB2_EPP1008_0001 : EPP1008_78E8D3DD;
    {attribute addProperty Name "RC20_AB6 (EPP1008-0001)"}
    {attribute addProperty PreviousPort "RC20_AB2 (EPP1008-0001) : B"}
    {attribute addProperty SyncUnit "C20"}
    RC20_AB6_EPP1008_0001 : EPP1008_78E8D3DD;
    {attribute addProperty Name "RC20_AB3 (EPP1008-0001)"}
    {attribute addProperty PreviousPort "RC20_AB6 (EPP1008-0001) : B"}
    {attribute addProperty SyncUnit "C20"}
    RC20_AB3_EPP1008_0001 : EPP1008_78E8D3DD;
    {attribute addProperty Name "RC20_AB4 (EPP1008-0001)"}
    {attribute addProperty PreviousPort "RC20_AB3 (EPP1008-0001) : B"}
    {attribute addProperty SyncUnit "C20"}
    RC20_AB4_EPP1008_0001 : EPP1008_78E8D3DD;
    {attribute addProperty Name "RC20_AB7 (EPP1008-0001)"}
    {attribute addProperty PreviousPort "RC20_EPP (EPP1322-0001) : B"}
    {attribute addProperty SyncUnit "C20"}
    RC20_AB7_EPP1008_0001 : EPP1008_78E8D3DD;
    {attribute addProperty Name "RC20_AB9 (EPP1008-0001)"}
    {attribute addProperty PreviousPort "RC20_AB7 (EPP1008-0001) : B"}
    {attribute addProperty SyncUnit "C20"}
    RC20_AB9_EPP1008_0001 : EPP1008_78E8D3DD;
    {attribute addProperty Name "RC20_AB10 (EPP1008-0001)"}
    {attribute addProperty PreviousPort "RC20_AB9 (EPP1008-0001) : B"}
    {attribute addProperty SyncUnit "C20"}
    RC20_AB10_EPP1008_0001 : EPP1008_78E8D3DD;
    {attribute addProperty Name "RC20_AB8 (EPP1008-0001)"}
    {attribute addProperty PreviousPort "RC20_AB10 (EPP1008-0001) : B"}
    {attribute addProperty SyncUnit "C20"}
    RC20_AB8_EPP1008_0001 : EPP1008_78E8D3DD;
    {attribute addProperty Name "RC20_AB5 (EPP1008-0001)"}
    {attribute addProperty PreviousPort "RC20_AB8 (EPP1008-0001) : B"}
    {attribute addProperty SyncUnit "C20"}
    RC20_AB5_EPP1008_0001 : EPP1008_78E8D3DD;
END_STRUCT
END_TYPE

// ---- DUTs/IO/Topology/RC20_A3_EK1122_1263CE61.TcDUT
{attribute 'GeneratedUsingTerminal: EK1122-0000-0018'}
{attribute addProperty BoxType "EK1122-0000-0018"}
{attribute addProperty Id "RC20_EPP_EPP1322_0001RC20_EPP_EPP1322_0001_59D450BA120"}
{attribute addProperty CRC "308530785"}
{attribute addProperty Size "120"}
{attribute addProperty Name "RC20_A3 (EK1122)"}
TYPE RC20_A3_EK1122_1263CE61 EXTENDS EK1122_1FC0878B :
STRUCT
    {attribute addProperty Name "RC20_EPP (EPP1322-0001)"}
    {attribute addProperty PreviousPort "RC20_A3 (EK1122) : D"}
    {attribute addProperty SyncUnit "default"}
    RC20_EPP_EPP1322_0001 : RC20_EPP_EPP1322_0001_59D450BA;
END_STRUCT
END_TYPE

// ---- DUTs/IO/Topology/RC20_1_EK1100_F221D0A9.TcDUT
{attribute 'GeneratedUsingTerminal: EK1100-0000-0018'}
{attribute addProperty BoxType "EK1100-0000-0018"}
{attribute addProperty Id "RC20_A2_EK1122RC20_A2_EK1122_77321D6773RC20_A3_EK1122RC20_A3_EK1122_1263CE61120RC20_A5_EL1809EL1809_32157CFD20RC20_A6_EL1809EL1809_32157CFD20RC20_A7_EL2809EL2809_2B6483BD19RC20_A8_EL2809EL2809_2B6483BD19RC20_A9_EL2809EL2809_2B6483BD19RC20_1_EndTerminal_EL9010EL9010_D29C20850"}
{attribute addProperty CRC "4062302377"}
{attribute addProperty Size "290"}
{attribute addProperty Name "RC20_1 (EK1100)"}
TYPE RC20_1_EK1100_F221D0A9 EXTENDS EK1100_1FC0878B :
STRUCT
    {attribute addProperty Name "RC20_A2 (EK1122)"}
    {attribute addProperty PreviousPort "RC20_1 (EK1100) : B"}
    {attribute addProperty SyncUnit "default"}
    RC20_A2_EK1122 : RC20_A2_EK1122_77321D67;
    {attribute addProperty Name "RC20_A3 (EK1122)"}
    {attribute addProperty PreviousPort "RC20_A2 (EK1122) : C"}
    {attribute addProperty SyncUnit "default"}
    RC20_A3_EK1122 : RC20_A3_EK1122_1263CE61;
    {attribute addProperty Name "RC20_A5 (EL1809)"}
    {attribute addProperty PreviousPort "RC20_A3 (EK1122) : C"}
    {attribute addProperty SyncUnit "C20"}
    RC20_A5_EL1809 : EL1809_32157CFD;
    {attribute addProperty Name "RC20_A6 (EL1809)"}
    {attribute addProperty PreviousPort "RC20_A5 (EL1809) : B"}
    {attribute addProperty SyncUnit "C20"}
    RC20_A6_EL1809 : EL1809_32157CFD;
    {attribute addProperty Name "RC20_A7 (EL2809)"}
    {attribute addProperty PreviousPort "RC20_A6 (EL1809) : B"}
    {attribute addProperty SyncUnit "C20"}
    RC20_A7_EL2809 : EL2809_2B6483BD;
    {attribute addProperty Name "RC20_A8 (EL2809)"}
    {attribute addProperty PreviousPort "RC20_A7 (EL2809) : B"}
    {attribute addProperty SyncUnit "C20"}
    RC20_A8_EL2809 : EL2809_2B6483BD;
    {attribute addProperty Name "RC20_A9 (EL2809)"}
    {attribute addProperty PreviousPort "RC20_A8 (EL2809) : B"}
    {attribute addProperty SyncUnit "C20"}
    RC20_A9_EL2809 : EL2809_2B6483BD;
    {attribute addProperty Name "RC20_1_EndTerminal (EL9010)"}
    {attribute addProperty PreviousPort "RC20_A9 (EL2809) : B"}
    {attribute addProperty SyncUnit "default"}
    RC20_1_EndTerminal_EL9010 : EL9010_D29C2085;
END_STRUCT
END_TYPE

// ---- DUTs/IO/Topology/RC20_2_EK1100_5EABB509.TcDUT
{attribute 'GeneratedUsingTerminal: EK1100-0000-0018'}
{attribute addProperty BoxType "EK1100-0000-0018"}
{attribute addProperty Id "RC20_B1_EL7041_1000EL7041_86DE63E743RC20_B2_EL7041_1000EL7041_86DE63E743RC20_C11_EL7041_1000EL7041_86DE63E743RC20_C12_EL7041_1000EL7041_86DE63E743RC20_C21_EL7041_1000EL7041_86DE63E743RC20_C22_EL7041_1000EL7041_86DE63E743RC20_2_EndTerminal_EL9010EL9010_D29C20850"}
{attribute addProperty CRC "1588311305"}
{attribute addProperty Size "258"}
{attribute addProperty Name "RC20_2 (EK1100)"}
TYPE RC20_2_EK1100_5EABB509 EXTENDS EK1100_1FC0878B :
STRUCT
    {attribute addProperty Name "RC20_B1 (EL7041-1000)"}
    {attribute addProperty PreviousPort "RC20_2 (EK1100) : B"}
    {attribute addProperty SyncUnit "C20"}
    RC20_B1_EL7041_1000 : EL7041_86DE63E7;
    {attribute addProperty Name "RC20_B2 (EL7041-1000)"}
    {attribute addProperty PreviousPort "RC20_B1 (EL7041-1000) : B"}
    {attribute addProperty SyncUnit "C20"}
    RC20_B2_EL7041_1000 : EL7041_86DE63E7;
    {attribute addProperty Name "RC20_C11 (EL7041-1000)"}
    {attribute addProperty PreviousPort "RC20_B2 (EL7041-1000) : B"}
    {attribute addProperty SyncUnit "C20"}
    RC20_C11_EL7041_1000 : EL7041_86DE63E7;
    {attribute addProperty Name "RC20_C12 (EL7041-1000)"}
    {attribute addProperty PreviousPort "RC20_C11 (EL7041-1000) : B"}
    {attribute addProperty SyncUnit "C20"}
    RC20_C12_EL7041_1000 : EL7041_86DE63E7;
    {attribute addProperty Name "RC20_C21 (EL7041-1000)"}
    {attribute addProperty PreviousPort "RC20_C12 (EL7041-1000) : B"}
    {attribute addProperty SyncUnit "C20"}
    RC20_C21_EL7041_1000 : EL7041_86DE63E7;
    {attribute addProperty Name "RC20_C22 (EL7041-1000)"}
    {attribute addProperty PreviousPort "RC20_C21 (EL7041-1000) : B"}
    {attribute addProperty SyncUnit "C20"}
    RC20_C22_EL7041_1000 : EL7041_86DE63E7;
    {attribute addProperty Name "RC20_2_EndTerminal (EL9010)"}
    {attribute addProperty PreviousPort "RC20_C22 (EL7041-1000) : B"}
    {attribute addProperty SyncUnit "default"}
    RC20_2_EndTerminal_EL9010 : EL9010_D29C2085;
END_STRUCT
END_TYPE

// ---- DUTs/IO/Topology/R8_A8_EK1122_2533F93A.TcDUT
{attribute 'GeneratedUsingTerminal: EK1122-0000-0018'}
{attribute addProperty BoxType "EK1122-0000-0018"}
{attribute addProperty Id "RC10_1_EK1100RC10_1_EK1100_40BAEC0F290RC10_2_EK1100RC10_2_EK1100_27865421258RC20_1_EK1100RC20_1_EK1100_F221D0A9290RC20_2_EK1100RC20_2_EK1100_5EABB509258"}
{attribute addProperty CRC "624163130"}
{attribute addProperty Size "1096"}
{attribute addProperty Name "R8_A8 (EK1122)"}
TYPE R8_A8_EK1122_2533F93A EXTENDS EK1122_1FC0878B :
STRUCT
    {attribute addProperty Name "RC10_1 (EK1100)"}
    {attribute addProperty PreviousPort "R8_A8 (EK1122) : D"}
    {attribute addProperty SyncUnit "default"}
    RC10_1_EK1100 : RC10_1_EK1100_40BAEC0F;
    {attribute addProperty Name "RC10_2 (EK1100)"}
    {attribute addProperty PreviousPort "RC10_1 (EK1100) : C"}
    {attribute addProperty SyncUnit "default"}
    RC10_2_EK1100 : RC10_2_EK1100_27865421;
    {attribute addProperty Name "RC20_1 (EK1100)"}
    {attribute addProperty PreviousPort "R8_A8 (EK1122) : B"}
    {attribute addProperty SyncUnit "default"}
    RC20_1_EK1100 : RC20_1_EK1100_F221D0A9;
    {attribute addProperty Name "RC20_2 (EK1100)"}
    {attribute addProperty PreviousPort "RC20_1 (EK1100) : C"}
    {attribute addProperty SyncUnit "default"}
    RC20_2_EK1100 : RC20_2_EK1100_5EABB509;
END_STRUCT
END_TYPE

// ---- DUTs/IO/Topology/RC30_A2_EK1122_334E4763.TcDUT
{attribute 'GeneratedUsingTerminal: EK1122-0000-0018'}
{attribute addProperty BoxType "EK1122-0000-0018"}
{attribute addProperty Id "RC30_VI_AES_D_BC_ECAT_xAES_A3B0707168RC30_SAFETY_Flexi_Soft_EtherCAT_GatewayFlexi_Soft_EtherCAT_Gateway_DE394EDD5"}
{attribute addProperty CRC "860768099"}
{attribute addProperty Size "73"}
{attribute addProperty Name "RC30_A2 (EK1122)"}
TYPE RC30_A2_EK1122_334E4763 EXTENDS EK1122_1FC0878B :
STRUCT
    {attribute addProperty Name "RC30_VI (AES-D-BC-ECAT)"}
    {attribute addProperty PreviousPort "RC30_A2 (EK1122) : D"}
    {attribute addProperty SyncUnit "C30"}
    RC30_VI_AES_D_BC_ECAT_x : AES_A3B07071;
    {attribute addProperty Name "RC30_SAFETY (Flexi Soft EtherCAT Gateway)"}
    {attribute addProperty PreviousPort "RC30_A2 (EK1122) : B"}
    {attribute addProperty SyncUnit "C30"}
    RC30_SAFETY_Flexi_Soft_EtherCAT_Gateway : Flexi_Soft_EtherCAT_Gateway_DE394EDD;
END_STRUCT
END_TYPE

// ---- DUTs/IO/Topology/RC30_EPP_EPP1322_0001_EDDD6881.TcDUT
{attribute 'GeneratedUsingTerminal: EPP1322-0001-0017'}
{attribute addProperty BoxType "EPP1322-0001-0017"}
{attribute addProperty Id "RC30_AB1_EPP1008_0001EPP1008_78E8D3DD12RC30_AB2_EPP1008_0001EPP1008_78E8D3DD12RC30_AB6_EPP1008_0001EPP1008_78E8D3DD12RC30_AB3_EPP1008_0001EPP1008_78E8D3DD12RC30_AB4_EPP1008_0001EPP1008_78E8D3DD12RC30_AB7_EPP1008_0001EPP1008_78E8D3DD12RC30_AB9_EPP1008_0001EPP1008_78E8D3DD12RC30_AB10_EPP1008_0001EPP1008_78E8D3DD12RC30_AB8_EPP1008_0001EPP1008_78E8D3DD12RC30_AB5_EPP1008_0001EPP1008_78E8D3DD12"}
{attribute addProperty CRC "3990710401"}
{attribute addProperty Size "120"}
{attribute addProperty Name "RC30_EPP (EPP1322-0001)"}
TYPE RC30_EPP_EPP1322_0001_EDDD6881 EXTENDS EPP1322_1FC0878B :
STRUCT
    {attribute addProperty Name "RC30_AB1 (EPP1008-0001)"}
    {attribute addProperty PreviousPort "RC30_EPP (EPP1322-0001) : D"}
    {attribute addProperty SyncUnit "C30"}
    RC30_AB1_EPP1008_0001 : EPP1008_78E8D3DD;
    {attribute addProperty Name "RC30_AB2 (EPP1008-0001)"}
    {attribute addProperty PreviousPort "RC30_AB1 (EPP1008-0001) : B"}
    {attribute addProperty SyncUnit "C30"}
    RC30_AB2_EPP1008_0001 : EPP1008_78E8D3DD;
    {attribute addProperty Name "RC30_AB6 (EPP1008-0001)"}
    {attribute addProperty PreviousPort "RC30_AB2 (EPP1008-0001) : B"}
    {attribute addProperty SyncUnit "C30"}
    RC30_AB6_EPP1008_0001 : EPP1008_78E8D3DD;
    {attribute addProperty Name "RC30_AB3 (EPP1008-0001)"}
    {attribute addProperty PreviousPort "RC30_AB6 (EPP1008-0001) : B"}
    {attribute addProperty SyncUnit "C30"}
    RC30_AB3_EPP1008_0001 : EPP1008_78E8D3DD;
    {attribute addProperty Name "RC30_AB4 (EPP1008-0001)"}
    {attribute addProperty PreviousPort "RC30_AB3 (EPP1008-0001) : B"}
    {attribute addProperty SyncUnit "C30"}
    RC30_AB4_EPP1008_0001 : EPP1008_78E8D3DD;
    {attribute addProperty Name "RC30_AB7 (EPP1008-0001)"}
    {attribute addProperty PreviousPort "RC30_EPP (EPP1322-0001) : B"}
    {attribute addProperty SyncUnit "C30"}
    RC30_AB7_EPP1008_0001 : EPP1008_78E8D3DD;
    {attribute addProperty Name "RC30_AB9 (EPP1008-0001)"}
    {attribute addProperty PreviousPort "RC30_AB7 (EPP1008-0001) : B"}
    {attribute addProperty SyncUnit "C30"}
    RC30_AB9_EPP1008_0001 : EPP1008_78E8D3DD;
    {attribute addProperty Name "RC30_AB10 (EPP1008-0001)"}
    {attribute addProperty PreviousPort "RC30_AB9 (EPP1008-0001) : B"}
    {attribute addProperty SyncUnit "C30"}
    RC30_AB10_EPP1008_0001 : EPP1008_78E8D3DD;
    {attribute addProperty Name "RC30_AB8 (EPP1008-0001)"}
    {attribute addProperty PreviousPort "RC30_AB10 (EPP1008-0001) : B"}
    {attribute addProperty SyncUnit "C30"}
    RC30_AB8_EPP1008_0001 : EPP1008_78E8D3DD;
    {attribute addProperty Name "RC30_AB5 (EPP1008-0001)"}
    {attribute addProperty PreviousPort "RC30_AB8 (EPP1008-0001) : B"}
    {attribute addProperty SyncUnit "C30"}
    RC30_AB5_EPP1008_0001 : EPP1008_78E8D3DD;
END_STRUCT
END_TYPE

// ---- DUTs/IO/Topology/RC30_A3_EK1122_482A08F6.TcDUT
{attribute 'GeneratedUsingTerminal: EK1122-0000-0018'}
{attribute addProperty BoxType "EK1122-0000-0018"}
{attribute addProperty Id "RC30_EPP_EPP1322_0001RC30_EPP_EPP1322_0001_EDDD6881120"}
{attribute addProperty CRC "1210714358"}
{attribute addProperty Size "120"}
{attribute addProperty Name "RC30_A3 (EK1122)"}
TYPE RC30_A3_EK1122_482A08F6 EXTENDS EK1122_1FC0878B :
STRUCT
    {attribute addProperty Name "RC30_EPP (EPP1322-0001)"}
    {attribute addProperty PreviousPort "RC30_A3 (EK1122) : D"}
    {attribute addProperty SyncUnit "default"}
    RC30_EPP_EPP1322_0001 : RC30_EPP_EPP1322_0001_EDDD6881;
END_STRUCT
END_TYPE

// ---- DUTs/IO/Topology/RC30_1_EK1100_B995809E.TcDUT
{attribute 'GeneratedUsingTerminal: EK1100-0000-0018'}
{attribute addProperty BoxType "EK1100-0000-0018"}
{attribute addProperty Id "RC30_A2_EK1122RC30_A2_EK1122_334E476373RC30_A3_EK1122RC30_A3_EK1122_482A08F6120RC30_A5_EL1809EL1809_32157CFD20RC30_A6_EL1809EL1809_32157CFD20RC30_A7_EL2809EL2809_2B6483BD19RC30_A8_EL2809EL2809_2B6483BD19RC30_A9_EL2809EL2809_2B6483BD19RC30_1_EndTerminal_EL9010EL9010_D29C20850"}
{attribute addProperty CRC "3113582750"}
{attribute addProperty Size "290"}
{attribute addProperty Name "RC30_1 (EK1100)"}
TYPE RC30_1_EK1100_B995809E EXTENDS EK1100_1FC0878B :
STRUCT
    {attribute addProperty Name "RC30_A2 (EK1122)"}
    {attribute addProperty PreviousPort "RC30_1 (EK1100) : B"}
    {attribute addProperty SyncUnit "default"}
    RC30_A2_EK1122 : RC30_A2_EK1122_334E4763;
    {attribute addProperty Name "RC30_A3 (EK1122)"}
    {attribute addProperty PreviousPort "RC30_A2 (EK1122) : C"}
    {attribute addProperty SyncUnit "default"}
    RC30_A3_EK1122 : RC30_A3_EK1122_482A08F6;
    {attribute addProperty Name "RC30_A5 (EL1809)"}
    {attribute addProperty PreviousPort "RC30_A3 (EK1122) : C"}
    {attribute addProperty SyncUnit "C30"}
    RC30_A5_EL1809 : EL1809_32157CFD;
    {attribute addProperty Name "RC30_A6 (EL1809)"}
    {attribute addProperty PreviousPort "RC30_A5 (EL1809) : B"}
    {attribute addProperty SyncUnit "C30"}
    RC30_A6_EL1809 : EL1809_32157CFD;
    {attribute addProperty Name "RC30_A7 (EL2809)"}
    {attribute addProperty PreviousPort "RC30_A6 (EL1809) : B"}
    {attribute addProperty SyncUnit "C30"}
    RC30_A7_EL2809 : EL2809_2B6483BD;
    {attribute addProperty Name "RC30_A8 (EL2809)"}
    {attribute addProperty PreviousPort "RC30_A7 (EL2809) : B"}
    {attribute addProperty SyncUnit "C30"}
    RC30_A8_EL2809 : EL2809_2B6483BD;
    {attribute addProperty Name "RC30_A9 (EL2809)"}
    {attribute addProperty PreviousPort "RC30_A8 (EL2809) : B"}
    {attribute addProperty SyncUnit "C30"}
    RC30_A9_EL2809 : EL2809_2B6483BD;
    {attribute addProperty Name "RC30_1_EndTerminal (EL9010)"}
    {attribute addProperty PreviousPort "RC30_A9 (EL2809) : B"}
    {attribute addProperty SyncUnit "default"}
    RC30_1_EndTerminal_EL9010 : EL9010_D29C2085;
END_STRUCT
END_TYPE

// ---- DUTs/IO/Topology/RC30_2_EK1100_8A0FE17C.TcDUT
{attribute 'GeneratedUsingTerminal: EK1100-0000-0018'}
{attribute addProperty BoxType "EK1100-0000-0018"}
{attribute addProperty Id "RC30_B1_EL7041_1000EL7041_86DE63E743RC30_B2_EL7041_1000EL7041_86DE63E743RC30_C11_EL7041_1000EL7041_86DE63E743RC30_C12_EL7041_1000EL7041_86DE63E743RC30_C21_EL7041_1000EL7041_86DE63E743RC30_C22_EL7041_1000EL7041_86DE63E743RC30_2_EndTerminal_EL9010EL9010_D29C20850"}
{attribute addProperty CRC "2316296572"}
{attribute addProperty Size "258"}
{attribute addProperty Name "RC30_2 (EK1100)"}
TYPE RC30_2_EK1100_8A0FE17C EXTENDS EK1100_1FC0878B :
STRUCT
    {attribute addProperty Name "RC30_B1 (EL7041-1000)"}
    {attribute addProperty PreviousPort "RC30_2 (EK1100) : B"}
    {attribute addProperty SyncUnit "C30"}
    RC30_B1_EL7041_1000 : EL7041_86DE63E7;
    {attribute addProperty Name "RC30_B2 (EL7041-1000)"}
    {attribute addProperty PreviousPort "RC30_B1 (EL7041-1000) : B"}
    {attribute addProperty SyncUnit "C30"}
    RC30_B2_EL7041_1000 : EL7041_86DE63E7;
    {attribute addProperty Name "RC30_C11 (EL7041-1000)"}
    {attribute addProperty PreviousPort "RC30_B2 (EL7041-1000) : B"}
    {attribute addProperty SyncUnit "C30"}
    RC30_C11_EL7041_1000 : EL7041_86DE63E7;
    {attribute addProperty Name "RC30_C12 (EL7041-1000)"}
    {attribute addProperty PreviousPort "RC30_C11 (EL7041-1000) : B"}
    {attribute addProperty SyncUnit "C30"}
    RC30_C12_EL7041_1000 : EL7041_86DE63E7;
    {attribute addProperty Name "RC30_C21 (EL7041-1000)"}
    {attribute addProperty PreviousPort "RC30_C12 (EL7041-1000) : B"}
    {attribute addProperty SyncUnit "C30"}
    RC30_C21_EL7041_1000 : EL7041_86DE63E7;
    {attribute addProperty Name "RC30_C22 (EL7041-1000)"}
    {attribute addProperty PreviousPort "RC30_C21 (EL7041-1000) : B"}
    {attribute addProperty SyncUnit "C30"}
    RC30_C22_EL7041_1000 : EL7041_86DE63E7;
    {attribute addProperty Name "RC30_2_EndTerminal (EL9010)"}
    {attribute addProperty PreviousPort "RC30_C22 (EL7041-1000) : B"}
    {attribute addProperty SyncUnit "default"}
    RC30_2_EndTerminal_EL9010 : EL9010_D29C2085;
END_STRUCT
END_TYPE

// ---- DUTs/IO/Topology/RC40_A2_EK1122_EAFADCC8.TcDUT
{attribute 'GeneratedUsingTerminal: EK1122-0000-0018'}
{attribute addProperty BoxType "EK1122-0000-0018"}
{attribute addProperty Id "RC40_VI_AES_D_BC_ECAT_xAES_A3B0707168RC40_SAFETY_Flexi_Soft_EtherCAT_GatewayFlexi_Soft_EtherCAT_Gateway_DE394EDD5"}
{attribute addProperty CRC "3942309064"}
{attribute addProperty Size "73"}
{attribute addProperty Name "RC40_A2 (EK1122)"}
TYPE RC40_A2_EK1122_EAFADCC8 EXTENDS EK1122_1FC0878B :
STRUCT
    {attribute addProperty Name "RC40_VI (AES-D-BC-ECAT)"}
    {attribute addProperty PreviousPort "RC40_A2 (EK1122) : D"}
    {attribute addProperty SyncUnit "C40"}
    RC40_VI_AES_D_BC_ECAT_x : AES_A3B07071;
    {attribute addProperty Name "RC40_SAFETY (Flexi Soft EtherCAT Gateway)"}
    {attribute addProperty PreviousPort "RC40_A2 (EK1122) : B"}
    {attribute addProperty SyncUnit "C40"}
    RC40_SAFETY_Flexi_Soft_EtherCAT_Gateway : Flexi_Soft_EtherCAT_Gateway_DE394EDD;
END_STRUCT
END_TYPE

// ---- DUTs/IO/Topology/RC40_EPP_EPP1322_0001_ECA1E6F9.TcDUT
{attribute 'GeneratedUsingTerminal: EPP1322-0001-0017'}
{attribute addProperty BoxType "EPP1322-0001-0017"}
{attribute addProperty Id "RC40_AB1_EPP1008_0001EPP1008_78E8D3DD12RC40_AB2_EPP1008_0001EPP1008_78E8D3DD12RC40_AB6_EPP1008_0001EPP1008_78E8D3DD12RC40_AB3_EPP1008_0001EPP1008_78E8D3DD12RC40_AB4_EPP1008_0001EPP1008_78E8D3DD12RC40_AB7_EPP1008_0001EPP1008_78E8D3DD12RC40_AB9_EPP1008_0001EPP1008_78E8D3DD12RC40_AB10_EPP1008_0001EPP1008_78E8D3DD12RC40_AB8_EPP1008_0001EPP1008_78E8D3DD12RC40_AB5_EPP1008_0001EPP1008_78E8D3DD12"}
{attribute addProperty CRC "3970033401"}
{attribute addProperty Size "120"}
{attribute addProperty Name "RC40_EPP (EPP1322-0001)"}
TYPE RC40_EPP_EPP1322_0001_ECA1E6F9 EXTENDS EPP1322_1FC0878B :
STRUCT
    {attribute addProperty Name "RC40_AB1 (EPP1008-0001)"}
    {attribute addProperty PreviousPort "RC40_EPP (EPP1322-0001) : D"}
    {attribute addProperty SyncUnit "C40"}
    RC40_AB1_EPP1008_0001 : EPP1008_78E8D3DD;
    {attribute addProperty Name "RC40_AB2 (EPP1008-0001)"}
    {attribute addProperty PreviousPort "RC40_AB1 (EPP1008-0001) : B"}
    {attribute addProperty SyncUnit "C40"}
    RC40_AB2_EPP1008_0001 : EPP1008_78E8D3DD;
    {attribute addProperty Name "RC40_AB6 (EPP1008-0001)"}
    {attribute addProperty PreviousPort "RC40_AB2 (EPP1008-0001) : B"}
    {attribute addProperty SyncUnit "C40"}
    RC40_AB6_EPP1008_0001 : EPP1008_78E8D3DD;
    {attribute addProperty Name "RC40_AB3 (EPP1008-0001)"}
    {attribute addProperty PreviousPort "RC40_AB6 (EPP1008-0001) : B"}
    {attribute addProperty SyncUnit "C40"}
    RC40_AB3_EPP1008_0001 : EPP1008_78E8D3DD;
    {attribute addProperty Name "RC40_AB4 (EPP1008-0001)"}
    {attribute addProperty PreviousPort "RC40_AB3 (EPP1008-0001) : B"}
    {attribute addProperty SyncUnit "C40"}
    RC40_AB4_EPP1008_0001 : EPP1008_78E8D3DD;
    {attribute addProperty Name "RC40_AB7 (EPP1008-0001)"}
    {attribute addProperty PreviousPort "RC40_EPP (EPP1322-0001) : B"}
    {attribute addProperty SyncUnit "C40"}
    RC40_AB7_EPP1008_0001 : EPP1008_78E8D3DD;
    {attribute addProperty Name "RC40_AB9 (EPP1008-0001)"}
    {attribute addProperty PreviousPort "RC40_AB7 (EPP1008-0001) : B"}
    {attribute addProperty SyncUnit "C40"}
    RC40_AB9_EPP1008_0001 : EPP1008_78E8D3DD;
    {attribute addProperty Name "RC40_AB10 (EPP1008-0001)"}
    {attribute addProperty PreviousPort "RC40_AB9 (EPP1008-0001) : B"}
    {attribute addProperty SyncUnit "C40"}
    RC40_AB10_EPP1008_0001 : EPP1008_78E8D3DD;
    {attribute addProperty Name "RC40_AB8 (EPP1008-0001)"}
    {attribute addProperty PreviousPort "RC40_AB10 (EPP1008-0001) : B"}
    {attribute addProperty SyncUnit "C40"}
    RC40_AB8_EPP1008_0001 : EPP1008_78E8D3DD;
    {attribute addProperty Name "RC40_AB5 (EPP1008-0001)"}
    {attribute addProperty PreviousPort "RC40_AB8 (EPP1008-0001) : B"}
    {attribute addProperty SyncUnit "C40"}
    RC40_AB5_EPP1008_0001 : EPP1008_78E8D3DD;
END_STRUCT
END_TYPE

